C05467=1236.826,137.681,-50.122,-177.956,5.568,148.362
C05468=1236.831,137.432,-50.101,-177.958,5.567,148.362
C05469=1236.835,137.183,-50.081,-177.961,5.566,148.363
C05470=1236.840,136.934,-50.061,-177.963,5.565,148.363
C05471=1236.845,136.684,-50.040,-177.966,5.564,148.364
C05472=1236.849,136.435,-50.019,-177.968,5.562,148.364
C05473=1236.855,136.186,-49.998,-177.971,5.562,148.365
C05474=1236.859,135.937,-49.978,-177.973,5.561,148.365
C05475=1236.864,135.688,-49.957,-177.976,5.560,148.366
C05476=1236.869,135.439,-49.937,-177.979,5.559,148.366
C05477=1236.873,135.190,-49.916,-177.981,5.558,148.367
C05478=1236.878,134.941,-49.895,-177.984,5.557,148.367
C05479=1236.883,134.692,-49.875,-177.986,5.555,148.368
C05480=1236.887,134.443,-49.854,-177.989,5.554,148.368
C05481=1236.893,134.174,-49.833,-177.991,5.554,148.369
C05482=1236.898,133.905,-49.810,-177.994,5.552,148.369
C05483=1236.903,133.636,-49.788,-177.997,5.551,148.370
C05484=1236.908,133.368,-49.767,-178.000,5.550,148.371
C05485=1236.913,133.119,-49.746,-178.002,5.549,148.371
C05486=1236.917,132.870,-49.725,-178.005,5.548,148.372
C05487=1236.922,132.621,-49.705,-178.007,5.548,148.372
C05488=1236.927,132.371,-49.685,-178.010,5.546,148.373
C05489=1236.932,132.122,-49.664,-178.012,5.545,148.373
C05490=1236.936,131.873,-49.644,-178.015,5.544,148.374
C05491=1236.941,131.624,-49.623,-178.018,5.543,148.374
C05492=1236.946,131.375,-49.602,-178.020,5.542,148.375
C05493=1236.951,131.125,-49.583,-178.022,5.541,148.375
C05494=1236.955,130.876,-49.562,-178.025,5.540,148.376
C05495=1236.960,130.627,-49.541,-178.028,5.539,148.376
C05496=1236.965,130.378,-49.521,-178.030,5.538,148.377
C05497=1236.970,130.129,-49.502,-178.032,5.537,148.377
C05498=1236.974,129.880,-49.481,-178.035,5.536,148.378
C05499=1236.979,129.631,-49.461,-178.038,5.535,148.379
C05500=1236.984,129.381,-49.441,-178.040,5.534,148.379
C05501=1236.989,129.132,-49.420,-178.043,5.533,148.380
C05502=1236.993,128.884,-49.400,-178.045,5.532,148.380
C05503=1236.998,128.635,-49.380,-178.048,5.531,148.381
C05504=1237.002,128.385,-49.360,-178.050,5.530,148.381
C05505=1237.008,128.136,-49.339,-178.053,5.529,148.382
C05506=1237.012,127.887,-49.319,-178.056,5.528,148.382
C05507=1237.017,127.638,-49.299,-178.058,5.527,148.383
C05508=1237.022,127.389,-49.279,-178.061,5.526,148.383
C05509=1237.027,127.139,-49.259,-178.063,5.525,148.384
C05510=1237.032,126.890,-49.238,-178.066,5.524,148.384
C05511=1237.036,126.641,-49.218,-178.069,5.523,148.385
C05512=1237.041,126.392,-49.198,-178.071,5.522,148.385
C05513=1237.045,126.143,-49.178,-178.073,5.521,148.386
C05514=1237.051,125.894,-49.159,-178.076,5.520,148.386
C05515=1237.055,125.645,-49.138,-178.078,5.520,148.387
C05516=1237.060,125.396,-49.118,-178.081,5.518,148.388
C05517=1237.064,125.146,-49.098,-178.083,5.517,148.388
C05518=1237.069,124.897,-49.077,-178.086,5.517,148.389
C05519=1237.074,124.648,-49.058,-178.089,5.516,148.389
C05520=1237.079,124.399,-49.038,-178.091,5.514,148.390
C05521=1237.084,124.150,-49.018,-178.094,5.513,148.390
C05522=1237.088,123.901,-48.998,-178.096,5.512,148.391
C05523=1237.093,123.651,-48.978,-178.099,5.512,148.391
C05524=1237.098,123.402,-48.958,-178.101,5.511,148.392
C05525=1237.102,123.153,-48.938,-178.104,5.509,148.392
C05526=1237.107,122.904,-48.918,-178.107,5.509,148.393
C05527=1237.112,122.655,-48.898,-178.109,5.508,148.394
C05528=1237.117,122.406,-48.878,-178.111,5.507,148.394
C05529=1237.121,122.156,-48.858,-178.114,5.506,148.395
C05530=1237.127,121.907,-48.839,-178.117,5.505,148.395
C05531=1237.131,121.659,-48.819,-178.119,5.504,148.396
C05532=1237.136,121.409,-48.799,-178.122,5.503,148.396
C05533=1237.140,121.160,-48.779,-178.124,5.502,148.397
C05534=1237.146,120.910,-48.758,-178.127,5.501,148.397
C05535=1237.151,120.661,-48.739,-178.130,5.500,148.398
C05536=1237.156,120.412,-48.719,-178.132,5.499,148.399
C05537=1237.160,120.163,-48.699,-178.134,5.499,148.399
C05538=1237.164,119.914,-48.679,-178.136,5.498,148.400
C05539=1237.169,119.665,-48.660,-178.140,5.496,148.400
C05540=1237.174,119.416,-48.640,-178.142,5.496,148.401
C05541=1237.179,119.167,-48.620,-178.144,5.495,148.401
C05542=1237.183,118.917,-48.600,-178.147,5.494,148.402
C05543=1237.189,118.668,-48.581,-178.150,5.493,148.403
C05544=1237.193,118.419,-48.561,-178.152,5.492,148.403
C05545=1237.198,118.170,-48.541,-178.155,5.491,148.404
C05546=1237.203,117.920,-48.521,-178.157,5.490,148.404
C05547=1237.208,117.671,-48.502,-178.160,5.489,148.405
C05548=1237.212,117.422,-48.482,-178.162,5.489,148.405
C05549=1237.217,117.173,-48.462,-178.165,5.488,148.406
C05550=1237.222,116.924,-48.443,-178.167,5.486,148.406
C05551=1237.227,116.674,-48.423,-178.170,5.486,148.407
C05552=1237.232,116.425,-48.403,-178.172,5.485,148.407
C05553=1237.237,116.177,-48.383,-178.175,5.484,148.408
C05554=1237.241,115.927,-48.364,-178.177,5.483,148.409
C05555=1237.246,115.678,-48.345,-178.180,5.482,148.409
C05556=1237.250,115.429,-48.324,-178.183,5.481,148.410
C05557=1237.255,115.180,-48.305,-178.185,5.480,148.410
C05558=1237.260,114.930,-48.285,-178.187,5.479,148.411
C05559=1237.265,114.681,-48.266,-178.190,5.479,148.411
C05560=1237.270,114.432,-48.246,-178.193,5.478,148.412
C05561=1237.275,114.182,-48.227,-178.195,5.476,148.412
C05562=1237.279,113.934,-48.207,-178.198,5.476,148.413
C05563=1237.284,113.685,-48.188,-178.201,5.475,148.414
C05564=1237.289,113.435,-48.168,-178.203,5.474,148.414
C05565=1237.294,113.186,-48.149,-178.205,5.473,148.415
C05566=1237.299,112.937,-48.129,-178.208,5.473,148.415
C05567=1237.303,112.688,-48.110,-178.210,5.472,148.416
C05568=1237.308,112.439,-48.091,-178.213,5.470,148.416
C05569=1237.313,112.189,-48.071,-178.216,5.470,148.417
C05570=1237.318,111.940,-48.051,-178.218,5.469,148.417
C05571=1237.323,111.691,-48.032,-178.221,5.468,148.418
C05572=1237.327,111.441,-48.013,-178.223,5.467,148.419
C05573=1237.332,111.193,-47.993,-178.226,5.467,148.419
C05574=1237.337,110.944,-47.973,-178.228,5.465,148.420
C05575=1237.342,110.694,-47.954,-178.231,5.464,148.420
C05576=1237.346,110.446,-47.935,-178.234,5.464,148.421
C05577=1237.351,110.196,-47.915,-178.236,5.463,148.421
C05578=1237.356,109.946,-47.896,-178.238,5.462,148.422
C05579=1237.361,109.698,-47.876,-178.241,5.461,148.423
C05580=1237.365,109.448,-47.857,-178.243,5.460,148.423
C05581=1237.370,109.199,-47.838,-178.246,5.459,148.424
C05582=1237.375,108.950,-47.818,-178.249,5.458,148.424
C05583=1237.381,108.700,-47.800,-178.251,5.457,148.425
C05584=1237.385,108.451,-47.781,-178.254,5.457,148.426
C05585=1237.390,108.182,-47.760,-178.256,5.456,148.426
C05586=1237.395,107.915,-47.739,-178.259,5.455,148.427
C05587=1237.400,107.646,-47.718,-178.262,5.454,148.427
C05588=1237.406,107.378,-47.697,-178.265,5.453,148.428
C05589=1237.411,107.128,-47.678,-178.267,5.452,148.428
C05590=1237.415,106.878,-47.659,-178.269,5.452,148.429
C05591=1237.420,106.630,-47.640,-178.273,5.450,148.430
C05592=1237.425,106.380,-47.620,-178.275,5.450,148.430
C05593=1237.429,106.131,-47.602,-178.277,5.449,148.431
C05594=1237.434,105.882,-47.582,-178.280,5.448,148.431
C05595=1237.439,105.633,-47.563,-178.283,5.447,148.432
C05596=1237.443,105.384,-47.544,-178.285,5.447,148.433
C05597=1237.449,105.134,-47.525,-178.287,5.446,148.433
C05598=1237.453,104.885,-47.506,-178.290,5.445,148.434
C05599=1237.458,104.636,-47.487,-178.293,5.443,148.434
C05600=1237.463,104.387,-47.467,-178.295,5.443,148.435
C05601=1237.468,104.138,-47.448,-178.298,5.442,148.436
C05602=1237.473,103.888,-47.429,-178.300,5.442,148.436
C05603=1237.477,103.639,-47.411,-178.303,5.441,148.437
C05604=1237.482,103.390,-47.391,-178.305,5.440,148.437
C05605=1237.488,103.141,-47.372,-178.308,5.439,148.438
C05606=1237.492,102.891,-47.353,-178.310,5.439,148.439
C05607=1237.497,102.642,-47.334,-178.313,5.438,148.439
C05608=1237.501,102.393,-47.315,-178.316,5.436,148.440
C05609=1237.507,102.144,-47.296,-178.318,5.436,148.440
C05610=1237.511,101.894,-47.277,-178.320,5.435,148.441
C05611=1237.516,101.645,-47.258,-178.323,5.434,148.441
C05612=1237.520,101.396,-47.239,-178.326,5.433,148.442
C05613=1237.526,101.146,-47.220,-178.328,5.433,148.443
C05614=1237.530,100.897,-47.201,-178.330,5.432,148.443
C05615=1237.535,100.648,-47.182,-178.333,5.431,148.444
C05616=1237.540,100.399,-47.164,-178.336,5.431,148.444
C05617=1237.545,100.150,-47.144,-178.338,5.430,148.445
C05618=1237.550,99.901,-47.126,-178.340,5.429,148.445
C05619=1237.555,99.651,-47.107,-178.344,5.428,148.446
C05620=1237.559,99.402,-47.088,-178.346,5.427,148.447
C05621=1237.564,99.153,-47.068,-178.348,5.426,148.447
C05622=1237.569,98.904,-47.050,-178.351,5.425,148.448
C05623=1237.574,98.655,-47.031,-178.354,5.425,148.448
C05624=1237.578,98.405,-47.013,-178.356,5.424,148.449
C05625=1237.584,98.156,-46.994,-178.358,5.423,148.449
C05626=1237.588,97.907,-46.974,-178.361,5.423,148.450
C05627=1237.593,97.657,-46.956,-178.364,5.422,148.451
C05628=1237.597,97.408,-46.937,-178.366,5.421,148.451
C05629=1237.602,97.159,-46.919,-178.368,5.420,148.452
C05630=1237.608,96.910,-46.900,-178.371,5.420,148.452
C05631=1237.612,96.660,-46.881,-178.374,5.418,148.453
C05632=1237.617,96.411,-46.862,-178.377,5.418,148.454
C05633=1237.622,96.162,-46.844,-178.379,5.417,148.454
C05634=1237.627,95.912,-46.824,-178.381,5.416,148.455
C05635=1237.632,95.663,-46.806,-178.384,5.415,148.455
C05636=1237.636,95.414,-46.787,-178.387,5.415,148.456
C05637=1237.642,95.165,-46.769,-178.389,5.414,148.457
C05638=1237.646,94.916,-46.750,-178.391,5.413,148.457
C05639=1237.651,94.666,-46.732,-178.394,5.413,148.458
C05640=1237.656,94.417,-46.712,-178.397,5.412,148.458
C05641=1237.661,94.168,-46.694,-178.399,5.411,148.459
C05642=1237.665,93.919,-46.675,-178.401,5.410,148.460
C05643=1237.670,93.669,-46.657,-178.404,5.410,148.460
C05644=1237.675,93.421,-46.638,-178.407,5.409,148.461
C05645=1237.679,93.171,-46.620,-178.409,5.409,148.461
C05646=1237.685,92.921,-46.601,-178.412,5.407,148.462
C05647=1237.690,92.673,-46.582,-178.415,5.406,148.463
C05648=1237.694,92.423,-46.564,-178.417,5.406,148.463
C05649=1237.700,92.173,-46.545,-178.420,5.405,148.464
C05650=1237.704,91.925,-46.527,-178.422,5.404,148.464
C05651=1237.708,91.675,-46.508,-178.425,5.403,148.465
C05652=1237.714,91.426,-46.489,-178.427,5.403,148.466
C05653=1237.719,91.177,-46.471,-178.430,5.402,148.466
C05654=1237.723,90.927,-46.453,-178.432,5.402,148.467
C05655=1237.728,90.679,-46.434,-178.435,5.401,148.467
C05656=1237.733,90.429,-46.416,-178.437,5.400,148.468
C05657=1237.738,90.179,-46.397,-178.440,5.399,148.469
C05658=1237.743,89.930,-46.379,-178.442,5.399,148.469
C05659=1237.747,89.681,-46.361,-178.445,5.398,148.470
C05660=1237.753,89.432,-46.342,-178.447,5.397,148.470
C05661=1237.757,89.182,-46.324,-178.450,5.397,148.471
C05662=1237.762,88.934,-46.305,-178.452,5.396,148.472
C05663=1237.767,88.684,-46.287,-178.455,5.395,148.472
C05664=1237.772,88.435,-46.268,-178.457,5.394,148.473
C05665=1237.777,88.185,-46.250,-178.460,5.394,148.473
C05666=1237.781,87.936,-46.231,-178.462,5.393,148.474
C05667=1237.786,87.687,-46.213,-178.465,5.393,148.475
C05668=1237.791,87.438,-46.195,-178.468,5.392,148.475
C05669=1237.796,87.188,-46.176,-178.470,5.391,148.476
C05670=1237.801,86.939,-46.158,-178.473,5.389,148.476
C05671=1237.806,86.690,-46.140,-178.476,5.389,148.477
C05672=1237.810,86.441,-46.122,-178.478,5.388,148.478
C05673=1237.815,86.191,-46.103,-178.481,5.388,148.478
C05674=1237.820,85.942,-46.085,-178.483,5.387,148.479
C05675=1237.825,85.692,-46.067,-178.486,5.386,148.479
C05676=1237.830,85.443,-46.049,-178.488,5.385,148.480
C05677=1237.835,85.193,-46.031,-178.491,5.385,148.481
C05678=1237.839,84.945,-46.012,-178.493,5.384,148.481
C05679=1237.844,84.696,-45.994,-178.496,5.383,148.482
C05680=1237.849,84.447,-45.976,-178.498,5.383,148.482
C05681=1237.854,84.197,-45.958,-178.501,5.382,148.483
C05682=1237.858,83.947,-45.940,-178.503,5.381,148.484
C05683=1237.864,83.698,-45.921,-178.506,5.381,148.484
C05684=1237.869,83.449,-45.903,-178.508,5.380,148.485
C05685=1237.874,83.200,-45.885,-178.511,5.379,148.486
C05686=1237.879,82.950,-45.867,-178.513,5.379,148.486
C05687=1237.883,82.701,-45.849,-178.516,5.378,148.487
C05688=1237.888,82.451,-45.831,-178.519,5.377,148.488
C05689=1237.893,82.183,-45.811,-178.521,5.377,148.488
C05690=1237.898,81.915,-45.792,-178.524,5.376,148.489
C05691=1237.904,81.646,-45.772,-178.527,5.376,148.489
C05692=1237.909,81.378,-45.753,-178.529,5.375,148.490
C05693=1237.914,81.129,-45.735,-178.532,5.374,148.491
C05694=1237.919,80.880,-45.717,-178.534,5.373,148.491
C05695=1237.924,80.631,-45.699,-178.537,5.373,148.492
C05696=1237.929,80.381,-45.681,-178.539,5.372,148.493
C05697=1237.933,80.131,-45.662,-178.542,5.372,148.493
C05698=1237.938,79.882,-45.644,-178.544,5.371,148.494
C05699=1237.943,79.633,-45.626,-178.547,5.370,148.495
C05700=1237.948,79.384,-45.608,-178.549,5.369,148.495
C05701=1237.953,79.135,-45.590,-178.552,5.369,148.496
C05702=1237.957,78.886,-45.572,-178.554,5.368,148.496
C05703=1237.962,78.636,-45.554,-178.557,5.368,148.497
C05704=1237.968,78.387,-45.537,-178.560,5.367,148.498
C05705=1237.972,78.137,-45.519,-178.562,5.366,148.498
C05706=1237.977,77.888,-45.501,-178.564,5.366,148.499
C05707=1237.982,77.638,-45.483,-178.567,5.365,148.499
C05708=1237.987,77.389,-45.465,-178.570,5.364,148.500
C05709=1237.992,77.140,-45.447,-178.572,5.364,148.501
C05710=1237.996,76.891,-45.429,-178.575,5.363,148.501
C05711=1238.001,76.642,-45.411,-178.578,5.362,148.502
C05712=1238.007,76.392,-45.394,-178.580,5.362,148.502
C05713=1238.011,76.143,-45.376,-178.582,5.361,148.503
C05714=1238.016,75.894,-45.358,-178.585,5.360,148.504
C05715=1238.021,75.645,-45.340,-178.588,5.360,148.504
C05716=1238.025,75.396,-45.322,-178.590,5.359,148.505
C05717=1238.031,75.146,-45.305,-178.593,5.359,148.506
C05718=1238.035,74.896,-45.287,-178.595,5.358,148.506
C05719=1238.040,74.647,-45.269,-178.598,5.357,148.507
C05720=1238.045,74.397,-45.251,-178.600,5.356,148.507
C05721=1238.050,74.148,-45.233,-178.603,5.356,148.508
C05722=1238.054,73.899,-45.216,-178.606,5.355,148.509
C05723=1238.059,73.650,-45.198,-178.608,5.355,148.509
C05724=1238.064,73.400,-45.180,-178.611,5.354,148.510
C05725=1238.069,73.151,-45.163,-178.613,5.353,148.510
C05726=1238.074,72.902,-45.145,-178.616,5.352,148.511
C05727=1238.079,72.652,-45.127,-178.618,5.352,148.512
C05728=1238.084,72.403,-45.109,-178.621,5.351,148.512
C05729=1238.088,72.154,-45.092,-178.623,5.351,148.513
C05730=1238.093,71.904,-45.074,-178.626,5.350,148.514
C05731=1238.098,71.655,-45.056,-178.628,5.350,148.514
C05732=1238.104,71.406,-45.039,-178.630,5.349,148.515
C05733=1238.108,71.156,-45.021,-178.633,5.349,148.516
C05734=1238.113,70.907,-45.003,-178.636,5.348,148.516
C05735=1238.118,70.658,-44.986,-178.638,5.347,148.517
C05736=1238.123,70.409,-44.968,-178.641,5.347,148.518
C05737=1238.128,70.159,-44.951,-178.643,5.346,148.518
C05738=1238.133,69.910,-44.933,-178.646,5.346,148.519
C05739=1238.137,69.661,-44.916,-178.648,5.345,148.519
C05740=1238.142,69.411,-44.899,-178.651,5.344,148.520
C05741=1238.147,69.162,-44.881,-178.653,5.344,148.521
C05742=1238.152,68.912,-44.863,-178.656,5.343,148.521
C05743=1238.157,68.663,-44.846,-178.659,5.342,148.522
C05744=1238.161,68.414,-44.828,-178.661,5.342,148.523
C05745=1238.167,68.164,-44.811,-178.664,5.341,148.523
C05746=1238.172,67.915,-44.793,-178.667,5.341,148.524
C05747=1238.176,67.665,-44.776,-178.669,5.340,148.524
C05748=1238.181,67.416,-44.758,-178.671,5.339,148.525
C05749=1238.186,67.166,-44.741,-178.673,5.339,148.526
C05750=1238.191,66.918,-44.724,-178.676,5.339,148.526
C05751=1238.196,66.668,-44.706,-178.679,5.338,148.527
C05752=1238.201,66.419,-44.688,-178.681,5.337,148.528
C05753=1238.206,66.170,-44.671,-178.684,5.337,148.528
C05754=1238.211,65.921,-44.654,-178.687,5.336,148.529
C05755=1238.216,65.671,-44.637,-178.689,5.335,148.529
C05756=1238.221,65.422,-44.619,-178.691,5.335,148.530
C05757=1238.225,65.172,-44.602,-178.694,5.334,148.531
C05758=1238.230,64.923,-44.584,-178.697,5.334,148.531
C05759=1238.235,64.673,-44.567,-178.699,5.333,148.532
C05760=1238.240,64.424,-44.550,-178.702,5.332,148.533
C05761=1238.245,64.175,-44.532,-178.704,5.332,148.533
C05762=1238.250,63.925,-44.515,-178.707,5.332,148.534
C05763=1238.255,63.677,-44.498,-178.709,5.331,148.535
C05764=1238.260,63.427,-44.480,-178.711,5.330,148.535
C05765=1238.264,63.177,-44.464,-178.714,5.330,148.536
C05766=1238.269,62.928,-44.446,-178.717,5.329,148.537
C05767=1238.274,62.678,-44.429,-178.719,5.329,148.537
C05768=1238.279,62.429,-44.411,-178.722,5.328,148.538
C05769=1238.284,62.180,-44.394,-178.724,5.328,148.539
C05770=1238.289,61.931,-44.378,-178.727,5.327,148.539
C05771=1238.294,61.682,-44.360,-178.730,5.326,148.540
C05772=1238.299,61.432,-44.342,-178.732,5.326,148.541
C05773=1238.304,61.182,-44.326,-178.735,5.325,148.541
C05774=1238.308,60.933,-44.308,-178.737,5.325,148.542
C05775=1238.313,60.684,-44.291,-178.739,5.324,148.542
C05776=1238.318,60.434,-44.274,-178.742,5.324,148.543
C05777=1238.323,60.185,-44.257,-178.744,5.323,148.544
C05778=1238.328,59.936,-44.239,-178.747,5.323,148.544
C05779=1238.333,59.686,-44.222,-178.750,5.322,148.545
C05780=1238.338,59.437,-44.206,-178.752,5.321,148.546
C05781=1238.343,59.188,-44.188,-178.755,5.321,148.546
C05782=1238.347,58.938,-44.171,-178.758,5.320,148.547
C05783=1238.353,58.689,-44.154,-178.760,5.320,148.548
C05784=1238.358,58.440,-44.137,-178.762,5.320,148.548
C05785=1238.363,58.190,-44.120,-178.764,5.319,148.549
C05786=1238.367,57.941,-44.103,-178.767,5.318,148.549
C05787=1238.372,57.691,-44.085,-178.770,5.318,148.550
C05788=1238.377,57.442,-44.069,-178.772,5.317,148.551
C05789=1238.382,57.192,-44.052,-178.775,5.317,148.551
C05790=1238.387,56.943,-44.035,-178.778,5.316,148.552
C05791=1238.392,56.694,-44.017,-178.780,5.315,148.553
C05792=1238.396,56.444,-44.001,-178.783,5.315,148.553
C05793=1238.402,56.176,-43.982,-178.786,5.314,148.554
C05794=1238.407,55.908,-43.964,-178.788,5.314,148.555
C05795=1238.413,55.639,-43.946,-178.791,5.313,148.555
C05796=1238.418,55.371,-43.928,-178.793,5.313,148.556
C05797=1238.423,55.121,-43.910,-178.796,5.312,148.557
C05798=1238.428,54.872,-43.894,-178.798,5.312,148.557
C05799=1238.432,54.623,-43.877,-178.801,5.312,148.558
C05800=1238.438,54.373,-43.860,-178.803,5.311,148.559
C05801=1238.442,54.124,-43.844,-178.806,5.310,148.559
C05802=1238.448,53.874,-43.827,-178.809,5.310,148.560
C05803=1238.452,53.625,-43.810,-178.811,5.309,148.561
C05804=1238.457,53.376,-43.793,-178.814,5.309,148.561
C05805=1238.462,53.126,-43.775,-178.817,5.308,148.562
C05806=1238.467,52.878,-43.759,-178.819,5.308,148.563
C05807=1238.472,52.628,-43.742,-178.821,5.307,148.563
C05808=1238.477,52.378,-43.725,-178.823,5.307,148.564
C05809=1238.482,52.129,-43.709,-178.826,5.306,148.565
C05810=1238.487,51.880,-43.691,-178.829,5.306,148.565
C05811=1238.491,51.630,-43.675,-178.831,5.305,148.566
C05812=1238.496,51.381,-43.658,-178.834,5.305,148.567
C05813=1238.502,51.132,-43.641,-178.836,5.305,148.567
C05814=1238.506,50.882,-43.625,-178.839,5.304,148.568
C05815=1238.511,50.633,-43.608,-178.841,5.304,148.569
C05816=1238.516,50.384,-43.591,-178.844,5.303,148.569
C05817=1238.521,50.134,-43.574,-178.847,5.302,148.570
C05818=1238.525,49.885,-43.558,-178.849,5.302,148.571
C05819=1238.531,49.635,-43.541,-178.852,5.301,148.571
C05820=1238.536,49.385,-43.525,-178.854,5.302,148.572
C05821=1238.540,49.136,-43.508,-178.857,5.301,148.573
C05822=1238.546,48.887,-43.491,-178.859,5.300,148.573
C05823=1238.551,48.637,-43.475,-178.861,5.299,148.574
C05824=1238.555,48.388,-43.458,-178.864,5.299,148.574
C05825=1238.560,48.139,-43.442,-178.867,5.298,148.575
C05826=1238.566,47.889,-43.424,-178.869,5.298,148.576
C05827=1238.570,47.640,-43.408,-178.871,5.298,148.576
C05828=1238.575,47.391,-43.391,-178.874,5.297,148.577
C05829=1238.580,47.141,-43.375,-178.877,5.297,148.578
C05830=1238.585,46.891,-43.358,-178.879,5.296,148.578
C05831=1238.590,46.642,-43.342,-178.882,5.296,148.579
C05832=1238.595,46.393,-43.325,-178.885,5.295,148.580
C05833=1238.599,46.143,-43.309,-178.887,5.295,148.580
C05834=1238.605,45.894,-43.292,-178.889,5.295,148.581
C05835=1238.610,45.644,-43.276,-178.892,5.294,148.582
C05836=1238.615,45.395,-43.259,-178.895,5.294,148.582
C05837=1238.619,45.146,-43.243,-178.897,5.293,148.583
C05838=1238.624,44.896,-43.226,-178.900,5.292,148.584
C05839=1238.630,44.647,-43.209,-178.902,5.292,148.584
C05840=1238.634,44.397,-43.193,-178.905,5.292,148.585
C05841=1238.639,44.148,-43.177,-178.907,5.291,148.586
C05842=1238.644,43.899,-43.160,-178.910,5.291,148.586
C05843=1238.648,43.649,-43.144,-178.912,5.290,148.587
C05844=1238.655,43.400,-43.127,-178.915,5.289,148.588
C05845=1238.659,43.150,-43.111,-178.917,5.289,148.588
C05846=1238.664,42.901,-43.094,-178.919,5.289,148.589
C05847=1238.669,42.652,-43.078,-178.922,5.288,148.590
C05848=1238.673,42.402,-43.062,-178.925,5.288,148.590
C05849=1238.678,42.153,-43.045,-178.927,5.287,148.591
C05850=1238.683,41.904,-43.029,-178.930,5.287,148.592
C05851=1238.689,41.654,-43.013,-178.932,5.287,148.592
C05852=1238.694,41.404,-42.996,-178.935,5.286,148.593
C05853=1238.699,41.156,-42.980,-178.937,5.286,148.594
C05854=1238.703,40.906,-42.964,-178.940,5.285,148.594
C05855=1238.708,40.656,-42.947,-178.942,5.285,148.595
C05856=1238.713,40.407,-42.931,-178.945,5.284,148.596
C05857=1238.718,40.157,-42.915,-178.947,5.284,148.596
C05858=1238.723,39.908,-42.898,-178.950,5.284,148.597
C05859=1238.727,39.659,-42.882,-178.952,5.283,148.598
C05860=1238.733,39.409,-42.866,-178.955,5.283,148.598
C05861=1238.738,39.160,-42.849,-178.958,5.282,148.599
C05862=1238.743,38.910,-42.833,-178.960,5.282,148.600
C05863=1238.748,38.661,-42.817,-178.962,5.282,148.600
C05864=1238.753,38.411,-42.801,-178.965,5.281,148.601
C05865=1238.758,38.162,-42.784,-178.968,5.281,148.602
C05866=1238.763,37.913,-42.768,-178.970,5.280,148.602
C05867=1238.768,37.663,-42.752,-178.973,5.279,148.603
C05868=1238.773,37.414,-42.736,-178.975,5.280,148.604
C05869=1238.777,37.164,-42.720,-178.978,5.279,148.604
C05870=1238.782,36.915,-42.704,-178.980,5.279,148.605
C05871=1238.787,36.665,-42.688,-178.983,5.278,148.606
C05872=1238.792,36.416,-42.671,-178.986,5.277,148.606
C05873=1238.797,36.166,-42.655,-178.988,5.278,148.607
C05874=1238.802,35.918,-42.639,-178.990,5.277,148.608
C05875=1238.807,35.667,-42.623,-178.993,5.277,148.609
C05876=1238.812,35.419,-42.607,-178.996,5.276,148.609
C05877=1238.817,35.169,-42.591,-178.998,5.275,148.610
C05878=1238.822,34.920,-42.575,-179.000,5.276,148.611
C05879=1238.827,34.670,-42.559,-179.003,5.275,148.611
C05880=1238.832,34.421,-42.542,-179.006,5.275,148.612
C05881=1238.837,34.171,-42.526,-179.008,5.274,148.613
C05882=1238.842,33.921,-42.511,-179.011,5.273,148.613
C05883=1238.847,33.673,-42.494,-179.013,5.273,148.614
C05884=1238.852,33.423,-42.479,-179.015,5.273,148.614
C05885=1238.857,33.174,-42.462,-179.018,5.272,148.615
C05886=1238.862,32.924,-42.446,-179.020,5.272,148.616
C05887=1238.866,32.675,-42.431,-179.023,5.272,148.616
C05888=1238.871,32.425,-42.415,-179.025,5.271,148.617
C05889=1238.876,32.176,-42.399,-179.028,5.271,148.618
C05890=1238.881,31.927,-42.383,-179.030,5.270,148.618
C05891=1238.886,31.677,-42.367,-179.033,5.270,148.619
C05892=1238.891,31.427,-42.351,-179.035,5.270,148.620
C05893=1238.896,31.178,-42.334,-179.038,5.269,148.621
C05894=1238.901,30.928,-42.319,-179.040,5.269,148.621
C05895=1238.907,30.679,-42.303,-179.043,5.268,148.622
C05896=1238.911,30.430,-42.287,-179.046,5.268,148.623
C05897=1238.916,30.161,-42.270,-179.048,5.268,148.623
C05898=1238.922,29.893,-42.253,-179.051,5.268,148.624
C05899=1238.927,29.624,-42.236,-179.054,5.267,148.625
C05900=1238.932,29.355,-42.219,-179.056,5.267,148.625
C05901=1238.937,29.106,-42.203,-179.059,5.266,148.626
C05902=1238.942,28.856,-42.187,-179.062,5.265,148.627
C05903=1238.947,28.607,-42.171,-179.064,5.265,148.628
C05904=1238.953,28.358,-42.155,-179.066,5.265,148.628
C05905=1238.957,28.108,-42.140,-179.069,5.265,148.629
C05906=1238.962,27.858,-42.124,-179.072,5.264,148.630
C05907=1238.967,27.610,-42.108,-179.074,5.263,148.630
C05908=1238.972,27.360,-42.092,-179.076,5.264,148.631
C05909=1238.977,27.110,-42.077,-179.079,5.263,148.632
C05910=1238.982,26.861,-42.062,-179.082,5.263,148.632
C05911=1238.987,26.612,-42.045,-179.084,5.262,148.633
C05912=1238.992,26.362,-42.029,-179.086,5.262,148.634
C05913=1238.997,26.113,-42.014,-179.089,5.262,148.634
C05914=1239.001,25.863,-41.998,-179.092,5.261,148.635
C05915=1239.007,25.614,-41.983,-179.094,5.261,148.636
C05916=1239.012,25.364,-41.967,-179.096,5.261,148.636
C05917=1239.017,25.115,-41.951,-179.099,5.260,148.637
C05918=1239.022,24.865,-41.935,-179.102,5.260,148.638
C05919=1239.027,24.616,-41.920,-179.104,5.259,148.638
C05920=1239.031,24.366,-41.904,-179.106,5.259,148.639
C05921=1239.037,24.117,-41.888,-179.109,5.259,148.640
C05922=1239.041,23.868,-41.873,-179.112,5.259,148.641
C05923=1239.046,23.617,-41.857,-179.115,5.258,148.641
C05924=1239.052,23.368,-41.842,-179.117,5.257,148.642
C05925=1239.057,23.119,-41.826,-179.119,5.258,148.643
C05926=1239.061,22.869,-41.810,-179.122,5.257,148.643
C05927=1239.066,22.620,-41.795,-179.125,5.257,148.644
C05928=1239.072,22.371,-41.779,-179.127,5.256,148.645
C05929=1239.076,22.122,-41.764,-179.129,5.256,148.645
C05930=1239.081,21.871,-41.748,-179.132,5.256,148.646
C05931=1239.086,21.622,-41.733,-179.135,5.255,148.647
C05932=1239.091,21.373,-41.718,-179.137,5.255,148.647
C05933=1239.096,21.124,-41.702,-179.139,5.255,148.648
C05934=1239.101,20.873,-41.686,-179.142,5.254,148.649
C05935=1239.106,20.624,-41.671,-179.145,5.254,148.650
C05936=1239.111,20.375,-41.655,-179.147,5.254,148.650
C05937=1239.116,20.125,-41.639,-179.149,5.254,148.651
C05938=1239.121,19.876,-41.624,-179.152,5.253,148.652
C05939=1239.126,19.626,-41.609,-179.155,5.252,148.652
C05940=1239.131,19.377,-41.593,-179.157,5.253,148.653
C05941=1239.136,19.128,-41.578,-179.159,5.252,148.654
C05942=1239.141,18.878,-41.562,-179.162,5.252,148.654
C05943=1239.146,18.628,-41.547,-179.165,5.251,148.655
C05944=1239.151,18.379,-41.532,-179.167,5.251,148.656
C05945=1239.156,18.130,-41.516,-179.170,5.251,148.656
C05946=1239.160,17.880,-41.501,-179.172,5.250,148.657
C05947=1239.166,17.631,-41.485,-179.175,5.250,148.658
C05948=1239.171,17.381,-41.471,-179.177,5.250,148.658
C05949=1239.176,17.132,-41.455,-179.180,5.249,148.659
C05950=1239.181,16.882,-41.440,-179.182,5.249,148.660
C05951=1239.186,16.632,-41.424,-179.185,5.248,148.660
C05952=1239.191,16.383,-41.409,-179.187,5.248,148.661
C05953=1239.196,16.134,-41.394,-179.190,5.248,148.662
C05954=1239.201,15.885,-41.378,-179.192,5.247,148.663
C05955=1239.206,15.635,-41.363,-179.194,5.248,148.663
C05956=1239.211,15.385,-41.348,-179.197,5.247,148.664
C05957=1239.216,15.135,-41.332,-179.200,5.247,148.665
C05958=1239.221,14.886,-41.317,-179.202,5.246,148.665
C05959=1239.226,14.637,-41.302,-179.204,5.246,148.666
C05960=1239.231,14.388,-41.287,-179.207,5.246,148.667
C05961=1239.236,14.138,-41.271,-179.210,5.246,148.668
C05962=1239.240,13.888,-41.257,-179.212,5.246,148.668
C05963=1239.246,13.638,-41.241,-179.215,5.245,148.669
C05964=1239.251,13.389,-41.226,-179.217,5.245,148.670
C05965=1239.256,13.140,-41.210,-179.220,5.244,148.670
C05966=1239.261,12.890,-41.196,-179.222,5.244,148.671
C05967=1239.266,12.641,-41.181,-179.225,5.244,148.672
C05968=1239.270,12.391,-41.165,-179.227,5.243,148.672
C05969=1239.276,12.142,-41.150,-179.230,5.244,148.673
C05970=1239.281,11.892,-41.135,-179.232,5.243,148.674
C05971=1239.285,11.643,-41.120,-179.235,5.242,148.674
C05972=1239.291,11.393,-41.105,-179.238,5.242,148.675
C05973=1239.295,11.144,-41.090,-179.240,5.242,148.676
C05974=1239.301,10.894,-41.075,-179.242,5.242,148.676
C05975=1239.306,10.645,-41.060,-179.245,5.241,148.677
C05976=1239.310,10.395,-41.044,-179.247,5.241,148.678
C05977=1239.315,10.145,-41.030,-179.250,5.241,148.679
C05978=1239.321,9.896,-41.014,-179.252,5.240,148.679
C05979=1239.325,9.647,-40.999,-179.255,5.240,148.680
C05980=1239.330,9.397,-40.985,-179.257,5.240,148.681
C05981=1239.336,9.148,-40.969,-179.260,5.239,148.681
C05982=1239.340,8.899,-40.954,-179.262,5.239,148.682
C05983=1239.346,8.649,-40.939,-179.265,5.240,148.683
C05984=1239.351,8.400,-40.924,-179.268,5.239,148.684
C05985=1239.355,8.151,-40.909,-179.270,5.238,148.684
C05986=1239.361,7.901,-40.895,-179.272,5.239,148.685
C05987=1239.365,7.651,-40.879,-179.275,5.238,148.686
C05988=1239.370,7.401,-40.865,-179.278,5.238,148.686
C05989=1239.376,7.152,-40.849,-179.280,5.237,148.687
C05990=1239.380,6.903,-40.834,-179.282,5.237,148.688
C05991=1239.385,6.653,-40.820,-179.285,5.237,148.688
C05992=1239.391,6.403,-40.804,-179.288,5.236,148.689
C05993=1239.395,6.154,-40.790,-179.290,5.237,148.690
C05994=1239.400,5.905,-40.775,-179.292,5.236,148.690
C05995=1239.406,5.655,-40.760,-179.295,5.235,148.691
C05996=1239.410,5.406,-40.745,-179.297,5.236,148.692
C05997=1239.415,5.156,-40.730,-179.300,5.235,148.692
C05998=1239.421,4.906,-40.715,-179.302,5.235,148.693
C05999=1239.425,4.657,-40.700,-179.304,5.235,148.694
C06000=1239.430,4.408,-40.686,-179.307,5.234,148.695
C06001=1239.436,4.138,-40.670,-179.310,5.234,148.695
C06002=1239.441,3.870,-40.654,-179.313,5.234,148.696
C06003=1239.447,3.601,-40.638,-179.316,5.233,148.697
C06004=1239.452,3.332,-40.622,-179.318,5.234,148.698
C06005=1239.457,3.083,-40.607,-179.321,5.233,148.698
C06006=1239.462,2.833,-40.593,-179.323,5.233,148.699
C06007=1239.467,2.584,-40.577,-179.325,5.233,148.700
C06008=1239.472,2.334,-40.563,-179.328,5.232,148.701
C06009=1239.477,2.085,-40.548,-179.331,5.232,148.701
C06010=1239.482,1.835,-40.534,-179.333,5.231,148.702
C06011=1239.488,1.585,-40.519,-179.336,5.232,148.703
C06012=1239.492,1.336,-40.504,-179.338,5.231,148.703
C06013=1239.497,1.086,-40.490,-179.341,5.231,148.704
C06014=1239.502,0.837,-40.475,-179.343,5.231,148.705
C06015=1239.508,0.587,-40.460,-179.346,5.230,148.705
C06016=1239.513,0.337,-40.445,-179.348,5.230,148.706
C06017=1239.517,0.088,-40.430,-179.350,5.230,148.707
C06018=1239.522,-0.161,-40.416,-179.353,5.229,148.707
C06019=1239.527,-0.410,-40.401,-179.356,5.229,148.708
C06020=1239.532,-0.660,-40.386,-179.358,5.230,148.709
C06021=1239.537,-0.910,-40.372,-179.361,5.229,148.710
C06022=1239.542,-1.159,-40.357,-179.363,5.228,148.710
C06023=1239.547,-1.409,-40.343,-179.366,5.229,148.711
C06024=1239.552,-1.659,-40.328,-179.368,5.228,148.712
C06025=1239.557,-1.907,-40.314,-179.371,5.228,148.712
C06026=1239.563,-2.157,-40.299,-179.373,5.228,148.713
C06027=1239.568,-2.407,-40.285,-179.376,5.227,148.714
C06028=1239.573,-2.657,-40.270,-179.378,5.227,148.715
C06029=1239.577,-2.906,-40.255,-179.380,5.227,148.715
C06030=1239.582,-3.155,-40.241,-179.383,5.227,148.716
C06031=1239.587,-3.405,-40.227,-179.386,5.226,148.717
C06032=1239.592,-3.654,-40.212,-179.388,5.226,148.717
C06033=1239.598,-3.904,-40.197,-179.390,5.226,148.718
C06034=1239.603,-4.154,-40.183,-179.394,5.226,148.719
C06035=1239.608,-4.404,-40.168,-179.396,5.226,148.720
C06036=1239.613,-4.653,-40.154,-179.398,5.225,148.720
C06037=1239.618,-4.902,-40.140,-179.401,5.225,148.721
C06038=1239.623,-5.151,-40.125,-179.403,5.225,148.722
C06039=1239.628,-5.401,-40.111,-179.406,5.225,148.722
C06040=1239.633,-5.651,-40.097,-179.408,5.225,148.723
C06041=1239.637,-5.900,-40.082,-179.410,5.224,148.724
C06042=1239.642,-6.150,-40.067,-179.413,5.224,148.724
C06043=1239.647,-6.399,-40.053,-179.415,5.224,148.725
C06044=1239.653,-6.649,-40.038,-179.418,5.224,148.726
C06045=1239.658,-6.899,-40.024,-179.420,5.223,148.727
C06046=1239.663,-7.148,-40.010,-179.422,5.223,148.727
C06047=1239.668,-7.397,-39.995,-179.425,5.223,148.728
C06048=1239.673,-7.647,-39.981,-179.428,5.223,148.729
C06049=1239.678,-7.897,-39.967,-179.430,5.223,148.730
C06050=1239.683,-8.146,-39.952,-179.433,5.222,148.730
C06051=1239.688,-8.396,-39.938,-179.436,5.222,148.731
C06052=1239.693,-8.646,-39.924,-179.438,5.222,148.732
C06053=1239.698,-8.895,-39.910,-179.440,5.222,148.732
C06054=1239.703,-9.144,-39.896,-179.443,5.221,148.733
C06055=1239.708,-9.394,-39.881,-179.445,5.221,148.734
C06056=1239.713,-9.643,-39.866,-179.448,5.221,148.734
C06057=1239.718,-9.893,-39.852,-179.450,5.220,148.735
C06058=1239.723,-10.143,-39.838,-179.453,5.221,148.736
C06059=1239.728,-10.392,-39.824,-179.455,5.220,148.736
C06060=1239.733,-10.641,-39.810,-179.457,5.220,148.737
C06061=1239.738,-10.891,-39.795,-179.460,5.220,148.738
C06062=1239.743,-11.141,-39.781,-179.463,5.220,148.739
C06063=1239.748,-11.390,-39.767,-179.465,5.220,148.739
C06064=1239.754,-11.639,-39.753,-179.468,5.219,148.740
C06065=1239.759,-11.889,-39.739,-179.470,5.219,148.741
C06066=1239.764,-12.139,-39.724,-179.473,5.219,148.742
C06067=1239.768,-12.388,-39.711,-179.475,5.219,148.742
C06068=1239.773,-12.638,-39.696,-179.478,5.218,148.743
C06069=1239.778,-12.887,-39.682,-179.480,5.218,148.744
C06070=1239.783,-13.137,-39.668,-179.483,5.218,148.744
C06071=1239.788,-13.386,-39.654,-179.485,5.218,148.745
C06072=1239.793,-13.636,-39.640,-179.487,5.218,148.746
C06073=1239.799,-13.885,-39.626,-179.491,5.218,148.747
C06074=1239.804,-14.135,-39.611,-179.493,5.218,148.747
C06075=1239.809,-14.385,-39.597,-179.495,5.217,148.748
C06076=1239.814,-14.634,-39.583,-179.498,5.217,148.749
C06077=1239.819,-14.884,-39.569,-179.500,5.217,148.749
C06078=1239.824,-15.133,-39.556,-179.503,5.217,148.750
C06079=1239.829,-15.383,-39.542,-179.505,5.217,148.751
C06080=1239.834,-15.633,-39.527,-179.507,5.216,148.751
C06081=1239.839,-15.882,-39.513,-179.510,5.216,148.752
C06082=1239.844,-16.131,-39.499,-179.512,5.216,148.753
C06083=1239.849,-16.381,-39.485,-179.515,5.216,148.754
C06084=1239.854,-16.631,-39.471,-179.517,5.215,148.754
C06085=1239.859,-16.880,-39.457,-179.520,5.216,148.755
C06086=1239.864,-17.130,-39.444,-179.523,5.215,148.756
C06087=1239.869,-17.380,-39.429,-179.525,5.215,148.757
C06088=1239.874,-17.629,-39.415,-179.527,5.215,148.757
C06089=1239.880,-17.878,-39.401,-179.530,5.214,148.758
C06090=1239.885,-18.128,-39.387,-179.532,5.215,148.759
C06091=1239.889,-18.377,-39.373,-179.535,5.214,148.759
C06092=1239.895,-18.627,-39.360,-179.537,5.214,148.760
C06093=1239.900,-18.877,-39.346,-179.540,5.214,148.761
C06094=1239.905,-19.127,-39.332,-179.542,5.213,148.761
C06095=1239.910,-19.376,-39.317,-179.544,5.214,148.762
C06096=1239.914,-19.625,-39.304,-179.547,5.213,148.763
C06097=1239.920,-19.875,-39.290,-179.550,5.213,148.764
C06098=1239.925,-20.125,-39.276,-179.552,5.213,148.764
C06099=1239.930,-20.374,-39.262,-179.555,5.213,148.765
C06100=1239.935,-20.624,-39.248,-179.557,5.213,148.766
C06101=1239.940,-20.874,-39.235,-179.560,5.213,148.767
C06102=1239.945,-21.123,-39.221,-179.562,5.212,148.767
C06103=1239.950,-21.372,-39.207,-179.564,5.212,148.768
C06104=1239.955,-21.622,-39.193,-179.567,5.212,148.769
C06105=1239.960,-21.891,-39.178,-179.570,5.212,148.770
C06106=1239.966,-22.160,-39.164,-179.572,5.212,148.770
C06107=1239.971,-22.429,-39.149,-179.575,5.211,148.771
C06108=1239.977,-22.699,-39.134,-179.578,5.211,148.772
C06109=1239.983,-22.948,-39.120,-179.580,5.212,148.773
C06110=1239.987,-23.198,-39.107,-179.583,5.211,148.773
C06111=1239.992,-23.448,-39.092,-179.585,5.211,148.774
C06112=1239.998,-23.697,-39.079,-179.588,5.211,148.775
C06113=1240.003,-23.947,-39.065,-179.590,5.210,148.775
C06114=1240.007,-24.196,-39.051,-179.592,5.211,148.776
C06115=1240.013,-24.446,-39.038,-179.595,5.210,148.777
C06116=1240.018,-24.696,-39.024,-179.598,5.210,148.777
C06117=1240.022,-24.944,-39.010,-179.600,5.210,148.778
C06118=1240.028,-25.195,-38.997,-179.602,5.209,148.779
C06119=1240.033,-25.444,-38.983,-179.605,5.210,148.780
C06120=1240.038,-25.694,-38.970,-179.608,5.209,148.780
C06121=1240.043,-25.943,-38.956,-179.610,5.209,148.781
C06122=1240.048,-26.192,-38.942,-179.612,5.209,148.782
C06123=1240.053,-26.442,-38.929,-179.615,5.209,148.783
C06124=1240.058,-26.692,-38.915,-179.617,5.209,148.783
C06125=1240.063,-26.941,-38.902,-179.620,5.209,148.784
C06126=1240.068,-27.191,-38.888,-179.622,5.208,148.785
C06127=1240.074,-27.441,-38.874,-179.624,5.208,148.785
C06128=1240.078,-27.690,-38.861,-179.627,5.208,148.786
C06129=1240.083,-27.940,-38.847,-179.629,5.208,148.787
C06130=1240.089,-28.190,-38.833,-179.632,5.208,148.788
C06131=1240.093,-28.439,-38.820,-179.635,5.207,148.788
C06132=1240.099,-28.689,-38.806,-179.637,5.208,148.789
C06133=1240.103,-28.938,-38.793,-179.640,5.207,148.790
C06134=1240.109,-29.188,-38.780,-179.642,5.208,148.790
C06135=1240.113,-29.437,-38.766,-179.645,5.207,148.791
C06136=1240.118,-29.687,-38.752,-179.647,5.207,148.792
C06137=1240.124,-29.936,-38.738,-179.649,5.207,148.793
C06138=1240.128,-30.186,-38.725,-179.652,5.206,148.793
C06139=1240.134,-30.436,-38.712,-179.654,5.207,148.794
C06140=1240.139,-30.685,-38.699,-179.657,5.206,148.795
C06141=1240.144,-30.935,-38.685,-179.659,5.207,148.796
C06142=1240.149,-31.184,-38.672,-179.662,5.206,148.796
C06143=1240.154,-31.434,-38.658,-179.665,5.206,148.797
C06144=1240.159,-31.683,-38.645,-179.667,5.206,148.798
C06145=1240.165,-31.933,-38.632,-179.669,5.206,148.798
C06146=1240.169,-32.183,-38.619,-179.671,5.206,148.799
C06147=1240.175,-32.432,-38.605,-179.674,5.205,148.800
C06148=1240.180,-32.682,-38.591,-179.676,5.206,148.800
C06149=1240.185,-32.931,-38.578,-179.679,5.205,148.801
C06150=1240.190,-33.181,-38.564,-179.681,5.205,148.802
C06151=1240.195,-33.431,-38.552,-179.684,5.205,148.803
C06152=1240.200,-33.680,-38.537,-179.687,5.205,148.803
C06153=1240.205,-33.930,-38.525,-179.689,5.205,148.804
C06154=1240.210,-34.180,-38.512,-179.691,5.205,148.805
C06155=1240.215,-34.429,-38.498,-179.694,5.205,148.806
C06156=1240.220,-34.679,-38.485,-179.696,5.204,148.806
C06157=1240.226,-34.928,-38.472,-179.699,5.204,148.807
C06158=1240.230,-35.178,-38.458,-179.701,5.204,148.808
C06159=1240.236,-35.427,-38.445,-179.704,5.204,148.808
C06160=1240.240,-35.677,-38.432,-179.706,5.204,148.809
C06161=1240.246,-35.926,-38.418,-179.708,5.203,148.810
C06162=1240.250,-36.177,-38.405,-179.712,5.203,148.811
C06163=1240.256,-36.426,-38.392,-179.714,5.204,148.811
C06164=1240.260,-36.676,-38.378,-179.716,5.203,148.812
C06165=1240.266,-36.925,-38.366,-179.718,5.203,148.813
C06166=1240.271,-37.174,-38.352,-179.721,5.203,148.814
C06167=1240.276,-37.425,-38.339,-179.723,5.203,148.814
C06168=1240.281,-37.674,-38.326,-179.726,5.203,148.815
C06169=1240.286,-37.924,-38.313,-179.728,5.203,148.816
C06170=1240.292,-38.173,-38.299,-179.731,5.202,148.816
C06171=1240.296,-38.423,-38.286,-179.733,5.202,148.817
C06172=1240.301,-38.672,-38.273,-179.736,5.203,148.818
C06173=1240.307,-38.922,-38.260,-179.738,5.202,148.819
C06174=1240.312,-39.172,-38.247,-179.741,5.202,148.819
C06175=1240.317,-39.421,-38.234,-179.743,5.202,148.820
C06176=1240.322,-39.671,-38.221,-179.745,5.202,148.821
C06177=1240.327,-39.920,-38.208,-179.748,5.202,148.821
C06178=1240.332,-40.170,-38.194,-179.751,5.201,148.822
C06179=1240.337,-40.420,-38.181,-179.753,5.202,148.823
C06180=1240.342,-40.669,-38.169,-179.755,5.201,148.824
C06181=1240.348,-40.919,-38.155,-179.757,5.201,148.824
C06182=1240.353,-41.168,-38.142,-179.761,5.201,148.825
C06183=1240.357,-41.419,-38.130,-179.763,5.202,148.826
C06184=1240.363,-41.668,-38.116,-179.765,5.201,148.827
C06185=1240.368,-41.917,-38.103,-179.767,5.201,148.827
C06186=1240.372,-42.167,-38.090,-179.770,5.201,148.828
C06187=1240.378,-42.416,-38.077,-179.773,5.200,148.829
C06188=1240.383,-42.666,-38.064,-179.775,5.201,148.829
C06189=1240.388,-42.916,-38.051,-179.778,5.200,148.830
C06190=1240.393,-43.165,-38.039,-179.780,5.200,148.831
C06191=1240.398,-43.415,-38.025,-179.782,5.200,148.831
C06192=1240.403,-43.665,-38.013,-179.784,5.200,148.832
C06193=1240.409,-43.914,-38.000,-179.788,5.200,148.833
C06194=1240.413,-44.163,-37.986,-179.790,5.200,148.834
C06195=1240.419,-44.413,-37.973,-179.792,5.200,148.835
C06196=1240.424,-44.662,-37.960,-179.795,5.199,148.835
C06197=1240.428,-44.912,-37.947,-179.797,5.200,148.836
C06198=1240.434,-45.162,-37.934,-179.800,5.199,148.837
C06199=1240.439,-45.411,-37.922,-179.802,5.200,148.837
C06200=1240.444,-45.661,-37.909,-179.804,5.199,148.838
C06201=1240.449,-45.911,-37.896,-179.807,5.199,148.839
C06202=1240.454,-46.160,-37.884,-179.809,5.199,148.839
C06203=1240.459,-46.410,-37.870,-179.812,5.200,148.840
C06204=1240.464,-46.660,-37.857,-179.814,5.199,148.841
C06205=1240.470,-46.909,-37.845,-179.817,5.199,148.842
C06206=1240.474,-47.159,-37.832,-179.819,5.199,148.842
C06207=1240.480,-47.409,-37.819,-179.822,5.198,148.843
C06208=1240.485,-47.658,-37.806,-179.824,5.199,148.844
C06209=1240.490,-47.928,-37.792,-179.827,5.198,148.845
C06210=1240.496,-48.198,-37.778,-179.829,5.199,148.846
C06211=1240.501,-48.467,-37.765,-179.832,5.198,148.846
C06212=1240.506,-48.737,-37.751,-179.835,5.198,148.847
C06213=1240.513,-48.987,-37.739,-179.837,5.198,148.848
C06214=1240.518,-49.236,-37.726,-179.840,5.198,148.849
C06215=1240.522,-49.486,-37.713,-179.842,5.198,148.849
C06216=1240.527,-49.735,-37.700,-179.845,5.198,148.850
C06217=1240.532,-49.985,-37.688,-179.847,5.198,148.851
C06218=1240.537,-50.235,-37.675,-179.849,5.198,148.851
C06219=1240.543,-50.484,-37.662,-179.852,5.197,148.852
C06220=1240.548,-50.734,-37.649,-179.854,5.198,148.853
C06221=1240.553,-50.983,-37.636,-179.857,5.197,148.853
C06222=1240.558,-51.234,-37.624,-179.859,5.197,148.854
C06223=1240.563,-51.483,-37.612,-179.861,5.197,148.855
C06224=1240.568,-51.732,-37.599,-179.864,5.198,148.856
C06225=1240.573,-51.982,-37.586,-179.867,5.197,148.857
C06226=1240.578,-52.232,-37.573,-179.869,5.197,148.857
C06227=1240.584,-52.481,-37.560,-179.871,5.197,148.858
C06228=1240.589,-52.731,-37.548,-179.874,5.197,148.859
C06229=1240.594,-52.981,-37.536,-179.876,5.197,148.859
C06230=1240.599,-53.231,-37.523,-179.878,5.197,148.860
C06231=1240.604,-53.480,-37.510,-179.881,5.197,148.861
C06232=1240.609,-53.729,-37.498,-179.883,5.197,148.861
C06233=1240.614,-53.979,-37.486,-179.886,5.196,148.862
C06234=1240.620,-54.228,-37.473,-179.888,5.196,148.863
C06235=1240.624,-54.478,-37.460,-179.891,5.197,148.864
C06236=1240.629,-54.728,-37.447,-179.894,5.196,148.865
C06237=1240.635,-54.978,-37.436,-179.896,5.196,148.865
C06238=1240.640,-55.227,-37.423,-179.898,5.196,148.866
C06239=1240.644,-55.477,-37.410,-179.900,5.196,148.867
C06240=1240.649,-55.726,-37.397,-179.903,5.196,148.867
C06241=1240.655,-55.976,-37.386,-179.905,5.196,148.868
C06242=1240.660,-56.226,-37.373,-179.908,5.196,148.869
C06243=1240.665,-56.475,-37.360,-179.910,5.196,148.869
C06244=1240.670,-56.726,-37.348,-179.913,5.195,148.870
C06245=1240.675,-56.975,-37.336,-179.915,5.196,148.871
C06246=1240.680,-57.224,-37.323,-179.918,5.196,148.872
C06247=1240.685,-57.473,-37.310,-179.920,5.196,148.873
C06248=1240.691,-57.723,-37.298,-179.923,5.195,148.873
C06249=1240.696,-57.973,-37.286,-179.925,5.196,148.874
C06250=1240.700,-58.223,-37.273,-179.927,5.195,148.875
C06251=1240.706,-58.473,-37.261,-179.930,5.196,148.875
C06252=1240.711,-58.722,-37.248,-179.932,5.195,148.876
C06253=1240.716,-58.972,-37.236,-179.935,5.195,148.877
C06254=1240.721,-59.221,-37.224,-179.937,5.195,148.877
C06255=1240.727,-59.471,-37.211,-179.940,5.194,148.878
C06256=1240.732,-59.721,-37.199,-179.942,5.195,148.879
C06257=1240.737,-59.971,-37.186,-179.945,5.195,148.880
C06258=1240.742,-60.220,-37.174,-179.947,5.195,148.880
C06259=1240.747,-60.470,-37.162,-179.950,5.194,148.881
C06260=1240.752,-60.719,-37.149,-179.952,5.195,148.882
C06261=1240.758,-60.969,-37.137,-179.954,5.194,148.883
C06262=1240.763,-61.218,-37.125,-179.956,5.195,148.883
C06263=1240.768,-61.468,-37.113,-179.959,5.194,148.884
C06264=1240.772,-61.718,-37.101,-179.961,5.194,148.885
C06265=1240.777,-61.967,-37.088,-179.964,5.194,148.885
C06266=1240.783,-62.217,-37.076,-179.966,5.194,148.886
C06267=1240.788,-62.467,-37.064,-179.969,5.194,148.887
C06268=1240.793,-62.717,-37.052,-179.971,5.194,148.888
C06269=1240.798,-62.966,-37.039,-179.974,5.194,148.888
C06270=1240.804,-63.216,-37.027,-179.976,5.194,148.889
C06271=1240.809,-63.465,-37.015,-179.979,5.194,148.890
C06272=1240.814,-63.715,-37.003,-179.981,5.194,148.891
C06273=1240.819,-63.964,-36.991,-179.983,5.194,148.891
C06274=1240.824,-64.214,-36.979,-179.986,5.194,148.892
C06275=1240.829,-64.464,-36.966,-179.988,5.194,148.893
C06276=1240.834,-64.714,-36.954,-179.990,5.194,148.893
C06277=1240.839,-64.963,-36.941,-179.993,5.193,148.894
C06278=1240.844,-65.213,-36.929,-179.995,5.194,148.895
C06279=1240.850,-65.463,-36.918,-179.998,5.193,148.896
C06280=1240.854,-65.712,-36.906,180.000,5.194,148.896
C06281=1240.860,-65.962,-36.894,179.997,5.193,148.897
C06282=1240.865,-66.211,-36.881,179.995,5.194,148.898
C06283=1240.870,-66.461,-36.869,179.992,5.193,148.899
C06284=1240.875,-66.711,-36.857,179.990,5.194,148.899
C06285=1240.880,-66.960,-36.845,179.988,5.193,148.900
C06286=1240.886,-67.210,-36.833,179.985,5.193,148.901
C06287=1240.891,-67.460,-36.821,179.983,5.193,148.901
C06288=1240.896,-67.709,-36.809,179.981,5.193,148.902
C06289=1240.901,-67.959,-36.796,179.978,5.193,148.903
C06290=1240.906,-68.208,-36.785,179.976,5.193,148.904
C06291=1240.911,-68.458,-36.773,179.973,5.193,148.904
C06292=1240.916,-68.708,-36.761,179.971,5.193,148.905
C06293=1240.922,-68.958,-36.749,179.968,5.193,148.906
C06294=1240.927,-69.208,-36.737,179.966,5.193,148.907
C06295=1240.932,-69.457,-36.725,179.963,5.193,148.907
C06296=1240.937,-69.706,-36.713,179.961,5.193,148.908
C06297=1240.943,-69.956,-36.701,179.958,5.193,148.909
C06298=1240.948,-70.206,-36.688,179.956,5.193,148.909
C06299=1240.952,-70.455,-36.677,179.954,5.192,148.910
C06300=1240.958,-70.705,-36.665,179.952,5.193,148.911
C06301=1240.963,-70.955,-36.653,179.949,5.192,148.912
C06302=1240.968,-71.204,-36.641,179.947,5.193,148.912
C06303=1240.973,-71.454,-36.629,179.944,5.192,148.913
C06304=1240.978,-71.704,-36.618,179.942,5.192,148.914
C06305=1240.984,-71.953,-36.605,179.939,5.192,148.914
C06306=1240.988,-72.203,-36.594,179.937,5.193,148.915
C06307=1240.994,-72.453,-36.582,179.934,5.192,148.916
C06308=1240.999,-72.703,-36.570,179.932,5.193,148.917
C06309=1241.004,-72.952,-36.558,179.929,5.192,148.917
C06310=1241.009,-73.202,-36.546,179.927,5.192,148.918
C06311=1241.014,-73.452,-36.534,179.925,5.192,148.919
C06312=1241.019,-73.701,-36.523,179.923,5.192,148.920
C06313=1241.024,-73.972,-36.510,179.920,5.192,148.920
C06314=1241.031,-74.242,-36.497,179.917,5.192,148.921
C06315=1241.036,-74.512,-36.484,179.915,5.192,148.922
C06316=1241.042,-74.782,-36.471,179.912,5.192,148.923
C06317=1241.046,-75.032,-36.459,179.910,5.192,148.923
C06318=1241.052,-75.281,-36.448,179.907,5.191,148.924
C06319=1241.058,-75.531,-36.436,179.905,5.192,148.925
C06320=1241.062,-75.780,-36.424,179.902,5.192,148.926
C06321=1241.068,-76.030,-36.412,179.900,5.192,148.926
C06322=1241.072,-76.280,-36.401,179.897,5.192,148.927
C06323=1241.078,-76.530,-36.389,179.895,5.192,148.928
C06324=1241.083,-76.780,-36.377,179.892,5.191,148.929
C06325=1241.088,-77.029,-36.366,179.890,5.192,148.929
C06326=1241.093,-77.279,-36.354,179.888,5.191,148.930
C06327=1241.098,-77.528,-36.342,179.886,5.192,148.931
C06328=1241.103,-77.778,-36.330,179.883,5.191,148.931
C06329=1241.109,-78.027,-36.318,179.881,5.191,148.932
C06330=1241.114,-78.277,-36.307,179.878,5.191,148.933
C06331=1241.119,-78.527,-36.295,179.876,5.191,148.934
C06332=1241.124,-78.777,-36.284,179.873,5.191,148.934
C06333=1241.129,-79.027,-36.272,179.871,5.191,148.935
C06334=1241.134,-79.276,-36.261,179.868,5.191,148.936
C06335=1241.140,-79.526,-36.249,179.866,5.191,148.937
C06336=1241.145,-79.776,-36.237,179.863,5.191,148.937
C06337=1241.150,-80.026,-36.226,179.861,5.191,148.938
C06338=1241.156,-80.275,-36.214,179.859,5.191,148.939
C06339=1241.160,-80.525,-36.203,179.856,5.191,148.939
C06340=1241.166,-80.774,-36.191,179.854,5.191,148.940
C06341=1241.170,-81.024,-36.180,179.852,5.191,148.941
C06342=1241.176,-81.274,-36.168,179.850,5.191,148.942
C06343=1241.181,-81.524,-36.157,179.847,5.191,148.942
C06344=1241.186,-81.774,-36.145,179.845,5.191,148.943
C06345=1241.191,-82.023,-36.134,179.842,5.191,148.944
C06346=1241.197,-82.272,-36.122,179.840,5.191,148.944
C06347=1241.201,-82.522,-36.111,179.837,5.191,148.945
C06348=1241.207,-82.772,-36.099,179.835,5.191,148.946
C06349=1241.212,-83.022,-36.087,179.833,5.191,148.947
C06350=1241.217,-83.272,-36.076,179.830,5.191,148.947
C06351=1241.222,-83.521,-36.065,179.827,5.191,148.948
C06352=1241.228,-83.770,-36.053,179.825,5.191,148.949
C06353=1241.232,-84.020,-36.041,179.823,5.191,148.950
C06354=1241.237,-84.270,-36.030,179.821,5.191,148.950
C06355=1241.243,-84.520,-36.018,179.818,5.190,148.951
C06356=1241.248,-84.769,-36.007,179.816,5.191,148.952
C06357=1241.253,-85.018,-35.995,179.813,5.190,148.952
C06358=1241.258,-85.268,-35.984,179.811,5.191,148.953
C06359=1241.263,-85.518,-35.972,179.808,5.190,148.954
C06360=1241.268,-85.768,-35.962,179.806,5.191,148.955
C06361=1241.274,-86.018,-35.950,179.804,5.190,148.955
C06362=1241.279,-86.267,-35.939,179.801,5.190,148.956
C06363=1241.284,-86.517,-35.928,179.799,5.190,148.957
C06364=1241.289,-86.767,-35.916,179.797,5.190,148.957
C06365=1241.294,-87.016,-35.904,179.795,5.191,148.958
C06366=1241.300,-87.266,-35.893,179.792,5.190,148.959
C06367=1241.305,-87.516,-35.882,179.790,5.191,148.960
C06368=1241.310,-87.765,-35.871,179.787,5.190,148.960
C06369=1241.315,-88.015,-35.859,179.785,5.191,148.961
C06370=1241.320,-88.264,-35.848,179.782,5.190,148.962
C06371=1241.325,-88.514,-35.837,179.780,5.191,148.963
C06372=1241.331,-88.765,-35.826,179.777,5.190,148.963
C06373=1241.335,-89.014,-35.815,179.775,5.191,148.964
C06374=1241.342,-89.263,-35.803,179.772,5.190,148.965
C06375=1241.346,-89.513,-35.792,179.770,5.190,148.965
C06376=1241.351,-89.763,-35.780,179.768,5.190,148.966
C06377=1241.357,-90.013,-35.769,179.765,5.190,148.967
C06378=1241.362,-90.262,-35.758,179.763,5.190,148.968
C06379=1241.367,-90.512,-35.747,179.761,5.190,148.968
C06380=1241.372,-90.762,-35.735,179.758,5.190,148.969
C06381=1241.377,-91.012,-35.725,179.756,5.190,148.970
C06382=1241.382,-91.261,-35.714,179.754,5.190,148.970
C06383=1241.388,-91.511,-35.702,179.751,5.190,148.971
C06384=1241.392,-91.760,-35.690,179.749,5.190,148.972
C06385=1241.398,-92.010,-35.680,179.746,5.190,148.973
C06386=1241.403,-92.260,-35.669,179.744,5.190,148.973
C06387=1241.408,-92.509,-35.657,179.742,5.190,148.974
C06388=1241.413,-92.760,-35.647,179.740,5.190,148.975
C06389=1241.418,-93.009,-35.636,179.737,5.190,148.975
C06390=1241.424,-93.259,-35.624,179.735,5.190,148.976
C06391=1241.429,-93.509,-35.613,179.732,5.190,148.977
C06392=1241.434,-93.758,-35.602,179.730,5.190,148.978
C06393=1241.439,-94.007,-35.591,179.727,5.190,148.979
C06394=1241.445,-94.258,-35.580,179.725,5.190,148.979
C06395=1241.450,-94.507,-35.569,179.722,5.190,148.980
C06396=1241.455,-94.756,-35.558,179.720,5.190,148.981
C06397=1241.460,-95.007,-35.547,179.718,5.190,148.981
C06398=1241.466,-95.256,-35.535,179.715,5.190,148.982
C06399=1241.471,-95.506,-35.525,179.713,5.190,148.983
C06400=1241.475,-95.756,-35.514,179.710,5.190,148.984
C06401=1241.481,-96.005,-35.503,179.708,5.190,148.984
C06402=1241.486,-96.255,-35.491,179.706,5.190,148.985
C06403=1241.491,-96.505,-35.480,179.704,5.190,148.986
C06404=1241.497,-96.755,-35.470,179.701,5.190,148.986
C06405=1241.501,-97.004,-35.459,179.699,5.190,148.987
C06406=1241.507,-97.254,-35.447,179.696,5.189,148.988
C06407=1241.512,-97.504,-35.437,179.694,5.190,148.988
C06408=1241.517,-97.753,-35.425,179.691,5.189,148.989
C06409=1241.522,-98.003,-35.415,179.689,5.190,148.990
C06410=1241.527,-98.252,-35.404,179.687,5.190,148.991
C06411=1241.532,-98.503,-35.393,179.685,5.190,148.991
C06412=1241.538,-98.752,-35.382,179.682,5.190,148.992
C06413=1241.543,-99.002,-35.371,179.680,5.190,148.993
C06414=1241.548,-99.252,-35.360,179.678,5.190,148.993
C06415=1241.554,-99.501,-35.350,179.675,5.189,148.994
C06416=1241.558,-99.751,-35.338,179.673,5.190,148.995
C06417=1241.564,-100.022,-35.326,179.670,5.189,148.996
C06418=1241.570,-100.293,-35.315,179.668,5.190,148.997
C06419=1241.575,-100.563,-35.303,179.665,5.190,148.997
C06420=1241.581,-100.834,-35.291,179.663,5.190,148.998
C06421=1241.587,-101.084,-35.281,179.660,5.189,148.999
C06422=1241.591,-101.334,-35.270,179.658,5.190,148.999
C06423=1241.597,-101.583,-35.259,179.655,5.189,149.000
C06424=1241.602,-101.833,-35.248,179.653,5.190,149.001
C06425=1241.607,-102.083,-35.237,179.651,5.189,149.002
C06426=1241.612,-102.332,-35.227,179.649,5.190,149.002
C06427=1241.618,-102.583,-35.215,179.646,5.189,149.003
C06428=1241.623,-102.831,-35.204,179.644,5.190,149.004
C06429=1241.628,-103.082,-35.194,179.641,5.189,149.004
C06430=1241.633,-103.331,-35.184,179.639,5.189,149.005
C06431=1241.638,-103.581,-35.172,179.637,5.190,149.006
C06432=1241.643,-103.831,-35.162,179.634,5.189,149.007
C06433=1241.648,-104.080,-35.151,179.632,5.190,149.007
C06434=1241.653,-104.330,-35.140,179.629,5.189,149.008
C06435=1241.659,-104.580,-35.130,179.627,5.190,149.009
C06436=1241.664,-104.829,-35.119,179.625,5.189,149.009
C06437=1241.669,-105.079,-35.109,179.623,5.190,149.010
C06438=1241.674,-105.329,-35.098,179.620,5.189,149.011
C06439=1241.680,-105.578,-35.087,179.618,5.189,149.012
C06440=1241.685,-105.828,-35.077,179.615,5.189,149.012
C06441=1241.690,-106.078,-35.066,179.613,5.189,149.013
C06442=1241.695,-106.328,-35.055,179.610,5.190,149.014
C06443=1241.701,-106.577,-35.045,179.608,5.190,149.015
C06444=1241.706,-106.827,-35.034,179.606,5.190,149.015
C06445=1241.711,-107.076,-35.023,179.603,5.190,149.016
C06446=1241.716,-107.327,-35.013,179.601,5.190,149.017
C06447=1241.721,-107.576,-35.003,179.598,5.189,149.018
C06448=1241.726,-107.826,-34.992,179.596,5.190,149.018
C06449=1241.732,-108.075,-34.981,179.593,5.189,149.019
C06450=1241.737,-108.325,-34.970,179.591,5.190,149.020
C06451=1241.742,-108.575,-34.960,179.589,5.189,149.020
C06452=1241.747,-108.825,-34.950,179.587,5.190,149.021
C06453=1241.753,-109.074,-34.939,179.585,5.190,149.022
C06454=1241.758,-109.324,-34.928,179.582,5.189,149.022
C06455=1241.763,-109.574,-34.918,179.580,5.189,149.023
C06456=1241.768,-109.824,-34.907,179.578,5.189,149.024
C06457=1241.773,-110.073,-34.896,179.575,5.189,149.024
C06458=1241.778,-110.323,-34.886,179.573,5.189,149.025
C06459=1241.784,-110.573,-34.876,179.571,5.189,149.026
C06460=1241.789,-110.823,-34.865,179.568,5.189,149.027
C06461=1241.795,-111.073,-34.855,179.566,5.189,149.027
C06462=1241.799,-111.322,-34.844,179.564,5.190,149.028
C06463=1241.805,-111.572,-34.833,179.561,5.189,149.029
C06464=1241.810,-111.822,-34.823,179.559,5.190,149.029
C06465=1241.816,-112.072,-34.813,179.556,5.189,149.030
C06466=1241.820,-112.321,-34.803,179.554,5.189,149.031
C06467=1241.825,-112.571,-34.792,179.552,5.189,149.032
C06468=1241.831,-112.820,-34.782,179.549,5.189,149.032
C06469=1241.836,-113.070,-34.771,179.547,5.189,149.033
C06470=1241.841,-113.320,-34.761,179.545,5.189,149.034
C06471=1241.846,-113.570,-34.750,179.543,5.190,149.034
C06472=1241.852,-113.820,-34.740,179.540,5.189,149.035
C06473=1241.857,-114.069,-34.730,179.538,5.190,149.036
C06474=1241.862,-114.319,-34.719,179.535,5.189,149.037
C06475=1241.867,-114.569,-34.710,179.533,5.189,149.037
C06476=1241.872,-114.818,-34.698,179.530,5.189,149.038
C06477=1241.878,-115.068,-34.688,179.528,5.189,149.039
C06478=1241.883,-115.317,-34.678,179.526,5.189,149.039
C06479=1241.888,-115.568,-34.667,179.523,5.189,149.040
C06480=1241.894,-115.817,-34.657,179.521,5.190,149.041
C06481=1241.899,-116.067,-34.646,179.519,5.189,149.042
C06482=1241.904,-116.317,-34.637,179.517,5.190,149.042
C06483=1241.909,-116.566,-34.627,179.514,5.189,149.043
C06484=1241.914,-116.816,-34.616,179.512,5.190,149.044
C06485=1241.920,-117.066,-34.606,179.509,5.189,149.044
C06486=1241.925,-117.316,-34.595,179.507,5.189,149.045
C06487=1241.930,-117.565,-34.586,179.504,5.189,149.046
C06488=1241.935,-117.815,-34.575,179.502,5.189,149.047
C06489=1241.940,-118.065,-34.565,179.500,5.190,149.047
C06490=1241.946,-118.315,-34.555,179.497,5.189,149.048
C06491=1241.952,-118.564,-34.544,179.495,5.190,149.049
C06492=1241.956,-118.814,-34.535,179.493,5.189,149.049
C06493=1241.961,-119.064,-34.524,179.491,5.190,149.050
C06494=1241.966,-119.314,-34.514,179.488,5.189,149.051
C06495=1241.972,-119.564,-34.504,179.486,5.189,149.052
C06496=1241.977,-119.813,-34.494,179.484,5.190,149.052
C06497=1241.982,-120.063,-34.483,179.481,5.189,149.053
C06498=1241.987,-120.313,-34.473,179.479,5.189,149.054
C06499=1241.993,-120.562,-34.463,179.477,5.189,149.054
C06500=1241.997,-120.812,-34.453,179.475,5.189,149.055
C06501=1242.003,-121.062,-34.443,179.472,5.189,149.056
C06502=1242.008,-121.311,-34.433,179.470,5.189,149.056
C06503=1242.014,-121.562,-34.423,179.467,5.189,149.057
C06504=1242.019,-121.811,-34.413,179.465,5.189,149.058
C06505=1242.024,-122.061,-34.403,179.463,5.190,149.059
C06506=1242.029,-122.311,-34.392,179.460,5.189,149.059
C06507=1242.034,-122.560,-34.383,179.458,5.189,149.060
C06508=1242.040,-122.810,-34.372,179.456,5.189,149.061
C06509=1242.045,-123.059,-34.362,179.453,5.189,149.061
C06510=1242.050,-123.310,-34.352,179.451,5.189,149.062
C06511=1242.055,-123.559,-34.343,179.449,5.189,149.063
C06512=1242.061,-123.809,-34.333,179.447,5.190,149.064
C06513=1242.066,-124.059,-34.322,179.444,5.189,149.064
C06514=1242.071,-124.309,-34.312,179.442,5.190,149.065
C06515=1242.077,-124.558,-34.302,179.439,5.189,149.066
C06516=1242.082,-124.808,-34.292,179.437,5.190,149.066
C06517=1242.087,-125.058,-34.283,179.434,5.189,149.067
C06518=1242.092,-125.308,-34.272,179.433,5.189,149.068
C06519=1242.098,-125.557,-34.262,179.430,5.189,149.068
C06520=1242.102,-125.807,-34.252,179.428,5.189,149.069
C06521=1241.681,-125.818,-34.287,179.424,5.193,149.071
C06522=1241.676,-125.568,-34.297,179.426,5.192,149.071
C06523=1241.670,-125.318,-34.306,179.428,5.193,149.070
C06524=1241.665,-125.068,-34.317,179.430,5.192,149.069
C06525=1241.660,-124.819,-34.327,179.433,5.193,149.068
C06526=1241.655,-124.569,-34.337,179.435,5.192,149.068
C06527=1241.649,-124.320,-34.347,179.437,5.193,149.067
C06528=1241.644,-124.069,-34.356,179.439,5.193,149.066
C06529=1241.639,-123.820,-34.367,179.442,5.192,149.066
C06530=1241.633,-123.570,-34.377,179.444,5.193,149.065
C06531=1241.629,-123.320,-34.387,179.446,5.192,149.064
C06532=1241.623,-123.071,-34.397,179.449,5.193,149.064
C06533=1241.618,-122.821,-34.407,179.451,5.193,149.063
C06534=1241.613,-122.571,-34.418,179.454,5.193,149.062
C06535=1241.608,-122.321,-34.427,179.456,5.193,149.061
C06536=1241.602,-122.071,-34.437,179.458,5.192,149.061
C06537=1241.596,-121.822,-34.447,179.461,5.193,149.060
C06538=1241.592,-121.572,-34.457,179.463,5.192,149.059
C06539=1241.587,-121.322,-34.467,179.465,5.193,149.059
C06540=1241.581,-121.073,-34.477,179.468,5.192,149.058
C06541=1241.576,-120.823,-34.488,179.470,5.193,149.057
C06542=1241.571,-120.573,-34.498,179.472,5.192,149.056
C06543=1241.566,-120.324,-34.508,179.475,5.193,149.056
C06544=1241.561,-120.074,-34.518,179.477,5.193,149.055
C06545=1241.555,-119.824,-34.529,179.479,5.192,149.054
C06546=1241.550,-119.575,-34.538,179.482,5.193,149.054
C06547=1241.545,-119.324,-34.549,179.483,5.193,149.053
C06548=1241.539,-119.074,-34.558,179.486,5.193,149.052
C06549=1241.534,-118.824,-34.569,179.488,5.193,149.052
C06550=1241.529,-118.575,-34.578,179.491,5.193,149.051
C06551=1241.524,-118.325,-34.589,179.493,5.193,149.050
C06552=1241.519,-118.075,-34.599,179.496,5.193,149.049
C06553=1241.513,-117.826,-34.609,179.498,5.193,149.049
C06554=1241.508,-117.576,-34.619,179.500,5.192,149.048
C06555=1241.503,-117.326,-34.630,179.503,5.193,149.047
C06556=1241.498,-117.077,-34.640,179.505,5.193,149.047
C06557=1241.492,-116.827,-34.650,179.507,5.193,149.046
C06558=1241.487,-116.577,-34.661,179.509,5.193,149.045
C06559=1241.482,-116.328,-34.671,179.512,5.193,149.044
C06560=1241.477,-116.078,-34.682,179.514,5.193,149.044
C06561=1241.472,-115.828,-34.692,179.516,5.192,149.043
C06562=1241.466,-115.579,-34.702,179.519,5.193,149.042
C06563=1241.461,-115.329,-34.713,179.521,5.192,149.042
C06564=1241.456,-115.079,-34.723,179.524,5.193,149.041
C06565=1241.451,-114.829,-34.733,179.526,5.193,149.040
C06566=1241.446,-114.580,-34.743,179.529,5.193,149.039
C06567=1241.440,-114.330,-34.753,179.531,5.193,149.039
C06568=1241.435,-114.080,-34.764,179.533,5.193,149.038
C06569=1241.430,-113.830,-34.774,179.535,5.193,149.037
C06570=1241.425,-113.580,-34.784,179.537,5.192,149.037
C06571=1241.419,-113.330,-34.795,179.540,5.193,149.036
C06572=1241.414,-113.081,-34.806,179.542,5.192,149.035
C06573=1241.409,-112.832,-34.816,179.545,5.193,149.034
C06574=1241.404,-112.582,-34.826,179.547,5.192,149.034
C06575=1241.399,-112.332,-34.836,179.550,5.193,149.033
C06576=1241.393,-112.082,-34.847,179.552,5.193,149.032
C06577=1241.388,-111.832,-34.857,179.555,5.193,149.032
C06578=1241.383,-111.582,-34.867,179.557,5.193,149.031
C06579=1241.378,-111.333,-34.879,179.559,5.192,149.030
C06580=1241.372,-111.083,-34.889,179.561,5.193,149.029
C06581=1241.367,-110.834,-34.899,179.563,5.192,149.029
C06582=1241.362,-110.583,-34.910,179.566,5.193,149.028
C06583=1241.356,-110.334,-34.920,179.568,5.192,149.027
C06584=1241.352,-110.084,-34.931,179.571,5.193,149.027
C06585=1241.346,-109.835,-34.941,179.573,5.193,149.026
C06586=1241.342,-109.585,-34.951,179.576,5.193,149.025
C06587=1241.336,-109.335,-34.962,179.578,5.193,149.024
C06588=1241.331,-109.085,-34.972,179.580,5.193,149.024
C06589=1241.326,-108.836,-34.983,179.583,5.193,149.023
C06590=1241.321,-108.586,-34.994,179.585,5.192,149.022
C06591=1241.315,-108.336,-35.004,179.587,5.193,149.022
C06592=1241.310,-108.086,-35.014,179.589,5.193,149.021
C06593=1241.305,-107.837,-35.025,179.592,5.193,149.020
C06594=1241.300,-107.587,-35.036,179.594,5.193,149.020
C06595=1241.294,-107.337,-35.046,179.596,5.193,149.019
C06596=1241.290,-107.088,-35.057,179.598,5.193,149.018
C06597=1241.284,-106.838,-35.068,179.601,5.193,149.017
C06598=1241.279,-106.588,-35.078,179.603,5.193,149.017
C06599=1241.273,-106.338,-35.088,179.605,5.193,149.016
C06600=1241.269,-106.089,-35.100,179.608,5.193,149.015
C06601=1241.263,-105.839,-35.110,179.610,5.193,149.015
C06602=1241.258,-105.589,-35.120,179.613,5.193,149.014
C06603=1241.253,-105.340,-35.131,179.615,5.193,149.013
C06604=1241.248,-105.090,-35.142,179.618,5.193,149.012
C06605=1241.242,-104.840,-35.152,179.620,5.193,149.012
C06606=1241.238,-104.591,-35.163,179.622,5.193,149.011
C06607=1241.232,-104.340,-35.175,179.625,5.193,149.010
C06608=1241.227,-104.091,-35.186,179.628,5.193,149.009
C06609=1241.222,-103.841,-35.196,179.630,5.193,149.009
C06610=1241.216,-103.591,-35.206,179.632,5.192,149.008
C06611=1241.211,-103.342,-35.218,179.634,5.193,149.007
C06612=1241.206,-103.092,-35.228,179.637,5.193,149.007
C06613=1241.201,-102.842,-35.238,179.639,5.193,149.006
C06614=1241.195,-102.593,-35.249,179.641,5.193,149.005
C06615=1241.190,-102.343,-35.260,179.644,5.193,149.004
C06616=1241.186,-102.093,-35.271,179.646,5.193,149.004
C06617=1241.180,-101.844,-35.281,179.649,5.193,149.003
C06618=1241.175,-101.594,-35.293,179.651,5.193,149.002
C06619=1241.170,-101.344,-35.303,179.654,5.193,149.002
C06620=1241.164,-101.095,-35.315,179.656,5.193,149.001
C06621=1241.159,-100.844,-35.325,179.658,5.193,149.000
C06622=1241.154,-100.574,-35.337,179.660,5.193,148.999
C06623=1241.148,-100.303,-35.348,179.663,5.194,148.999
C06624=1241.142,-100.032,-35.360,179.665,5.193,148.998
C06625=1241.137,-99.762,-35.372,179.668,5.193,148.997
C06626=1241.132,-99.512,-35.383,179.670,5.193,148.996
C06627=1241.126,-99.262,-35.394,179.673,5.193,148.996
C06628=1241.121,-99.013,-35.405,179.675,5.193,148.995
C06629=1241.116,-98.762,-35.416,179.678,5.193,148.994
C06630=1241.111,-98.513,-35.427,179.680,5.193,148.993
C06631=1241.106,-98.263,-35.437,179.683,5.194,148.993
C06632=1241.101,-98.014,-35.448,179.685,5.193,148.992
C06633=1241.095,-97.764,-35.459,179.687,5.193,148.991
C06634=1241.090,-97.514,-35.471,179.690,5.193,148.991
C06635=1241.085,-97.265,-35.481,179.692,5.193,148.990
C06636=1241.080,-97.015,-35.492,179.694,5.193,148.989
C06637=1241.075,-96.765,-35.503,179.696,5.193,148.988
C06638=1241.069,-96.515,-35.514,179.699,5.194,148.988
C06639=1241.064,-96.266,-35.525,179.701,5.193,148.987
C06640=1241.059,-96.016,-35.536,179.704,5.194,148.986
C06641=1241.054,-95.767,-35.547,179.706,5.193,148.986
C06642=1241.049,-95.516,-35.558,179.709,5.194,148.985
C06643=1241.043,-95.266,-35.569,179.711,5.193,148.984
C06644=1241.038,-95.018,-35.580,179.713,5.194,148.983
C06645=1241.033,-94.767,-35.591,179.715,5.193,148.983
C06646=1241.028,-94.518,-35.602,179.718,5.193,148.982
C06647=1241.022,-94.268,-35.613,179.720,5.194,148.981
C06648=1241.017,-94.018,-35.624,179.722,5.193,148.981
C06649=1241.013,-93.769,-35.636,179.725,5.194,148.980
C06650=1241.007,-93.519,-35.646,179.727,5.193,148.979
C06651=1241.002,-93.269,-35.658,179.730,5.194,148.978
C06652=1240.997,-93.019,-35.669,179.732,5.193,148.978
C06653=1240.991,-92.770,-35.679,179.735,5.194,148.977
C06654=1240.986,-92.520,-35.691,179.737,5.193,148.976
C06655=1240.981,-92.270,-35.702,179.740,5.194,148.975
C06656=1240.976,-92.021,-35.713,179.742,5.193,148.975
C06657=1240.971,-91.771,-35.724,179.745,5.194,148.974
C06658=1240.966,-91.521,-35.736,179.747,5.193,148.973
C06659=1240.961,-91.272,-35.747,179.749,5.194,148.973
C06660=1240.955,-91.022,-35.757,179.751,5.194,148.972
C06661=1240.950,-90.772,-35.769,179.754,5.193,148.971
C06662=1240.945,-90.523,-35.780,179.756,5.194,148.970
C06663=1240.940,-90.273,-35.792,179.758,5.193,148.970
C06664=1240.934,-90.023,-35.803,179.761,5.194,148.969
C06665=1240.929,-89.773,-35.814,179.763,5.193,148.968
C06666=1240.925,-89.524,-35.825,179.766,5.194,148.968
C06667=1240.919,-89.275,-35.837,179.768,5.194,148.967
C06668=1240.914,-89.024,-35.847,179.771,5.194,148.966
C06669=1240.909,-88.775,-35.858,179.773,5.194,148.965
C06670=1240.904,-88.525,-35.870,179.775,5.194,148.965
C06671=1240.898,-88.276,-35.881,179.777,5.194,148.964
C06672=1240.893,-88.026,-35.893,179.780,5.194,148.963
C06673=1240.888,-87.776,-35.904,179.782,5.194,148.963
C06674=1240.883,-87.526,-35.915,179.785,5.194,148.962
C06675=1240.878,-87.276,-35.927,179.787,5.194,148.961
C06676=1240.872,-87.027,-35.938,179.790,5.195,148.960
C06677=1240.868,-86.778,-35.949,179.792,5.194,148.960
C06678=1240.862,-86.528,-35.961,179.794,5.193,148.959
C06679=1240.857,-86.277,-35.972,179.797,5.194,148.958
C06680=1240.851,-86.028,-35.983,179.799,5.194,148.957
C06681=1240.847,-85.779,-35.994,179.802,5.194,148.957
C06682=1240.841,-85.529,-36.006,179.804,5.194,148.956
C06683=1240.836,-85.279,-36.018,179.806,5.194,148.955
C06684=1240.832,-85.029,-36.029,179.809,5.194,148.955
C06685=1240.826,-84.780,-36.040,179.811,5.194,148.954
C06686=1240.821,-84.530,-36.052,179.813,5.194,148.953
C06687=1240.815,-84.280,-36.063,179.816,5.194,148.952
C06688=1240.811,-84.030,-36.074,179.818,5.194,148.952
C06689=1240.805,-83.780,-36.086,179.821,5.195,148.951
C06690=1240.800,-83.531,-36.097,179.823,5.194,148.950
C06691=1240.794,-83.281,-36.109,179.826,5.195,148.950
C06692=1240.790,-83.032,-36.120,179.828,5.194,148.949
C06693=1240.785,-82.782,-36.131,179.830,5.195,148.948
C06694=1240.780,-82.532,-36.143,179.832,5.194,148.947
C06695=1240.775,-82.283,-36.155,179.835,5.195,148.947
C06696=1240.769,-82.033,-36.166,179.837,5.195,148.946
C06697=1240.764,-81.784,-36.177,179.840,5.195,148.945
C06698=1240.759,-81.534,-36.189,179.842,5.194,148.944
C06699=1240.754,-81.284,-36.201,179.845,5.195,148.944
C06700=1240.749,-81.034,-36.212,179.847,5.194,148.943
C06701=1240.744,-80.785,-36.224,179.849,5.194,148.942
C06702=1240.739,-80.535,-36.236,179.852,5.195,148.942
C06703=1240.733,-80.286,-36.247,179.854,5.194,148.941
C06704=1240.728,-80.036,-36.258,179.857,5.195,148.940
C06705=1240.722,-79.786,-36.270,179.859,5.194,148.939
C06706=1240.718,-79.536,-36.282,179.861,5.195,148.939
C06707=1240.712,-79.286,-36.294,179.864,5.195,148.938
C06708=1240.708,-79.037,-36.305,179.866,5.195,148.937
C06709=1240.702,-78.787,-36.317,179.868,5.195,148.937
C06710=1240.697,-78.537,-36.328,179.871,5.195,148.936
C06711=1240.691,-78.288,-36.339,179.873,5.195,148.935
C06712=1240.687,-78.039,-36.351,179.876,5.195,148.934
C06713=1240.682,-77.789,-36.363,179.878,5.195,148.934
C06714=1240.676,-77.539,-36.375,179.881,5.195,148.933
C06715=1240.672,-77.289,-36.387,179.883,5.195,148.932
C06716=1240.666,-77.040,-36.398,179.886,5.195,148.931
C06717=1240.661,-76.790,-36.410,179.888,5.195,148.931
C06718=1240.656,-76.540,-36.422,179.891,5.195,148.930
C06719=1240.651,-76.290,-36.433,179.893,5.195,148.929
C06720=1240.646,-76.040,-36.445,179.895,5.195,148.929
C06721=1240.640,-75.792,-36.457,179.897,5.195,148.928
C06722=1240.635,-75.542,-36.469,179.900,5.196,148.927
C06723=1240.630,-75.292,-36.480,179.902,5.195,148.926
C06724=1240.625,-75.042,-36.492,179.905,5.196,148.926
C06725=1240.620,-74.793,-36.503,179.907,5.195,148.925
C06726=1240.615,-74.522,-36.516,179.910,5.195,148.924
C06727=1240.609,-74.253,-36.529,179.912,5.195,148.923
C06728=1240.603,-73.982,-36.543,179.915,5.196,148.923
C06729=1240.597,-73.712,-36.555,179.918,5.196,148.922
C06730=1240.593,-73.462,-36.567,179.920,5.195,148.921
C06731=1240.587,-73.212,-36.579,179.923,5.196,148.920
C06732=1240.582,-72.962,-36.591,179.925,5.196,148.920
C06733=1240.577,-72.714,-36.602,179.928,5.196,148.919
C06734=1240.571,-72.464,-36.614,179.930,5.196,148.918
C06735=1240.566,-72.214,-36.626,179.932,5.196,148.917
C06736=1240.561,-71.964,-36.637,179.934,5.196,148.917
C06737=1240.556,-71.715,-36.650,179.937,5.196,148.916
C06738=1240.551,-71.465,-36.662,179.939,5.196,148.915
C06739=1240.546,-71.215,-36.673,179.942,5.196,148.915
C06740=1240.541,-70.966,-36.685,179.944,5.196,148.914
C06741=1240.535,-70.716,-36.697,179.947,5.197,148.913
C06742=1240.530,-70.466,-36.709,179.949,5.196,148.912
C06743=1240.525,-70.217,-36.721,179.952,5.196,148.912
C06744=1240.520,-69.967,-36.733,179.954,5.196,148.911
C06745=1240.515,-69.717,-36.745,179.957,5.196,148.910
C06746=1240.509,-69.467,-36.757,179.959,5.196,148.909
C06747=1240.505,-69.218,-36.769,179.961,5.197,148.909
C06748=1240.499,-68.969,-36.781,179.963,5.196,148.908
C06749=1240.494,-68.719,-36.793,179.966,5.197,148.907
C06750=1240.489,-68.469,-36.805,179.968,5.196,148.907
C06751=1240.484,-68.220,-36.817,179.971,5.197,148.906
C06752=1240.479,-67.970,-36.829,179.973,5.197,148.905
C06753=1240.474,-67.720,-36.841,179.976,5.197,148.904
C06754=1240.468,-67.470,-36.853,179.978,5.197,148.904
C06755=1240.463,-67.221,-36.866,179.981,5.197,148.903
C06756=1240.458,-66.972,-36.877,179.983,5.197,148.902
C06757=1240.453,-66.722,-36.889,179.986,5.197,148.901
C06758=1240.448,-66.472,-36.902,179.988,5.197,148.901
C06759=1240.443,-66.222,-36.914,179.990,5.197,148.900
C06760=1240.438,-65.972,-36.926,179.993,5.197,148.899
C06761=1240.433,-65.723,-36.938,179.995,5.197,148.899
C06762=1240.428,-65.473,-36.949,179.997,5.197,148.898
C06763=1240.423,-65.223,-36.962,180.000,5.197,148.897
C06764=1240.417,-64.973,-36.974,-179.998,5.197,148.896
C06765=1240.412,-64.724,-36.987,-179.995,5.198,148.896
C06766=1240.407,-64.474,-36.998,-179.993,5.197,148.895
C06767=1240.402,-64.225,-37.010,-179.990,5.197,148.894
C06768=1240.397,-63.975,-37.022,-179.988,5.197,148.893
C06769=1240.392,-63.726,-37.035,-179.985,5.198,148.893
C06770=1240.386,-63.476,-37.047,-179.983,5.197,148.892
C06771=1240.381,-63.227,-37.059,-179.980,5.198,148.891
C06772=1240.376,-62.976,-37.072,-179.978,5.197,148.891
C06773=1240.371,-62.727,-37.084,-179.976,5.198,148.890
C06774=1240.366,-62.477,-37.096,-179.974,5.198,148.889
C06775=1240.361,-62.228,-37.108,-179.971,5.198,148.888
C06776=1240.356,-61.978,-37.120,-179.969,5.198,148.888
C06777=1240.351,-61.729,-37.133,-179.966,5.198,148.887
C06778=1240.345,-61.479,-37.145,-179.964,5.198,148.886
C06779=1240.340,-61.229,-37.157,-179.961,5.198,148.885
C06780=1240.335,-60.980,-37.170,-179.959,5.198,148.885
C06781=1240.330,-60.729,-37.182,-179.956,5.198,148.884
C06782=1240.325,-60.480,-37.195,-179.954,5.198,148.883
C06783=1240.320,-60.230,-37.206,-179.951,5.198,148.883
C06784=1240.315,-59.981,-37.219,-179.949,5.199,148.882
C06785=1240.309,-59.731,-37.231,-179.947,5.199,148.881
C06786=1240.304,-59.482,-37.244,-179.944,5.199,148.880
C06787=1240.299,-59.232,-37.256,-179.942,5.199,148.880
C06788=1240.294,-58.982,-37.268,-179.939,5.199,148.879
C06789=1240.290,-58.733,-37.280,-179.937,5.199,148.878
C06790=1240.285,-58.483,-37.293,-179.935,5.199,148.878
C06791=1240.279,-58.233,-37.305,-179.932,5.199,148.877
C06792=1240.274,-57.984,-37.318,-179.929,5.199,148.876
C06793=1240.269,-57.734,-37.329,-179.927,5.199,148.875
C06794=1240.264,-57.485,-37.342,-179.925,5.199,148.875
C06795=1240.259,-57.235,-37.355,-179.922,5.199,148.874
C06796=1240.254,-56.985,-37.368,-179.920,5.199,148.873
C06797=1240.249,-56.735,-37.379,-179.918,5.199,148.873
C06798=1240.243,-56.486,-37.392,-179.915,5.200,148.872
C06799=1240.238,-56.237,-37.405,-179.913,5.199,148.871
C06800=1240.233,-55.986,-37.417,-179.910,5.200,148.870
C06801=1240.228,-55.737,-37.430,-179.908,5.199,148.870
C06802=1240.223,-55.488,-37.442,-179.905,5.200,148.869
C06803=1240.218,-55.238,-37.454,-179.903,5.199,148.868
C06804=1240.213,-54.988,-37.467,-179.900,5.200,148.867
C06805=1240.207,-54.738,-37.480,-179.898,5.200,148.867
C06806=1240.202,-54.489,-37.493,-179.895,5.200,148.866
C06807=1240.197,-54.239,-37.505,-179.893,5.200,148.865
C06808=1240.192,-53.989,-37.517,-179.891,5.200,148.865
C06809=1240.187,-53.740,-37.530,-179.888,5.201,148.864
C06810=1240.182,-53.490,-37.543,-179.886,5.200,148.863
C06811=1240.177,-53.241,-37.555,-179.883,5.201,148.862
C06812=1240.172,-52.991,-37.567,-179.881,5.200,148.862
C06813=1240.166,-52.741,-37.580,-179.878,5.201,148.861
C06814=1240.162,-52.491,-37.593,-179.876,5.200,148.860
C06815=1240.157,-52.242,-37.605,-179.873,5.201,148.859
C06816=1240.152,-51.993,-37.618,-179.871,5.200,148.859
C06817=1240.146,-51.743,-37.630,-179.869,5.201,148.858
C06818=1240.142,-51.493,-37.643,-179.866,5.201,148.857
C06819=1240.136,-51.243,-37.656,-179.864,5.201,148.857
C06820=1240.131,-50.994,-37.669,-179.861,5.202,148.856
C06821=1240.126,-50.745,-37.681,-179.859,5.201,148.855
C06822=1240.121,-50.495,-37.694,-179.856,5.202,148.854
C06823=1240.116,-50.245,-37.707,-179.854,5.201,148.854
C06824=1240.110,-49.995,-37.719,-179.851,5.202,148.853
C06825=1240.105,-49.746,-37.731,-179.849,5.201,148.852
C06826=1240.100,-49.496,-37.745,-179.846,5.202,148.851
C06827=1240.095,-49.246,-37.758,-179.844,5.201,148.851
C06828=1240.090,-48.997,-37.770,-179.842,5.202,148.850
C06829=1240.085,-48.748,-37.783,-179.840,5.202,148.849
C06830=1240.080,-48.478,-37.796,-179.837,5.202,148.849
C06831=1240.074,-48.208,-37.811,-179.834,5.202,148.848
C06832=1240.069,-47.938,-37.824,-179.832,5.202,148.847
C06833=1240.063,-47.669,-37.838,-179.829,5.202,148.846
C06834=1240.058,-47.419,-37.851,-179.826,5.203,148.846
C06835=1240.053,-47.170,-37.864,-179.824,5.202,148.845
C06836=1240.048,-46.920,-37.876,-179.821,5.203,148.844
C06837=1240.042,-46.671,-37.890,-179.819,5.202,148.843
C06838=1240.037,-46.421,-37.903,-179.816,5.203,148.843
C06839=1240.032,-46.171,-37.915,-179.814,5.203,148.842
C06840=1240.027,-45.922,-37.928,-179.812,5.203,148.841
C06841=1240.023,-45.672,-37.941,-179.809,5.203,148.840
C06842=1240.017,-45.422,-37.954,-179.807,5.203,148.840
C06843=1240.012,-45.173,-37.967,-179.804,5.204,148.839
C06844=1240.007,-44.923,-37.980,-179.802,5.203,148.838
C06845=1240.002,-44.674,-37.992,-179.799,5.204,148.838
C06846=1239.996,-44.424,-38.005,-179.797,5.203,148.837
C06847=1239.992,-44.174,-38.018,-179.794,5.204,148.836
C06848=1239.987,-43.925,-38.031,-179.792,5.203,148.835
C06849=1239.981,-43.675,-38.044,-179.789,5.204,148.835
C06850=1239.976,-43.425,-38.057,-179.787,5.204,148.834
C06851=1239.971,-43.176,-38.070,-179.785,5.204,148.833
C06852=1239.966,-42.926,-38.082,-179.782,5.205,148.832
C06853=1239.961,-42.676,-38.096,-179.780,5.204,148.832
C06854=1239.956,-42.427,-38.108,-179.777,5.205,148.831
C06855=1239.951,-42.177,-38.121,-179.775,5.205,148.830
C06856=1239.945,-41.928,-38.135,-179.772,5.205,148.830
C06857=1239.940,-41.678,-38.148,-179.770,5.204,148.829
C06858=1239.936,-41.428,-38.161,-179.767,5.205,148.828
C06859=1239.931,-41.179,-38.173,-179.765,5.205,148.827
C06860=1239.925,-40.929,-38.187,-179.762,5.205,148.827
C06861=1239.920,-40.679,-38.200,-179.760,5.206,148.826
C06862=1239.915,-40.430,-38.212,-179.758,5.205,148.825
C06863=1239.910,-40.180,-38.227,-179.755,5.206,148.825
C06864=1239.905,-39.931,-38.239,-179.753,5.205,148.824
C06865=1239.900,-39.681,-38.253,-179.750,5.206,148.823
C06866=1239.895,-39.431,-38.265,-179.748,5.206,148.822
C06867=1239.890,-39.182,-38.278,-179.745,5.206,148.821
C06868=1239.884,-38.932,-38.291,-179.743,5.205,148.821
C06869=1239.880,-38.683,-38.305,-179.740,5.206,148.820
C06870=1239.875,-38.433,-38.318,-179.738,5.207,148.819
C06871=1239.869,-38.183,-38.331,-179.736,5.206,148.819
C06872=1239.864,-37.934,-38.344,-179.733,5.207,148.818
C06873=1239.859,-37.684,-38.358,-179.731,5.206,148.817
C06874=1239.854,-37.435,-38.370,-179.728,5.207,148.817
C06875=1239.849,-37.185,-38.383,-179.726,5.207,148.816
C06876=1239.844,-36.935,-38.397,-179.723,5.207,148.815
C06877=1239.839,-36.686,-38.410,-179.721,5.208,148.814
C06878=1239.833,-36.436,-38.423,-179.718,5.207,148.814
C06879=1239.829,-36.186,-38.436,-179.715,5.207,148.813
C06880=1239.823,-35.937,-38.450,-179.713,5.207,148.812
C06881=1239.818,-35.688,-38.463,-179.711,5.208,148.811
C06882=1239.814,-35.438,-38.476,-179.709,5.207,148.811
C06883=1239.808,-35.188,-38.489,-179.706,5.208,148.810
C06884=1239.804,-34.939,-38.503,-179.703,5.208,148.809
C06885=1239.798,-34.689,-38.516,-179.701,5.208,148.809
C06886=1239.793,-34.439,-38.529,-179.699,5.209,148.808
C06887=1239.788,-34.190,-38.543,-179.696,5.208,148.807
C06888=1239.783,-33.940,-38.556,-179.694,5.209,148.807
C06889=1239.777,-33.691,-38.569,-179.691,5.208,148.806
C06890=1239.773,-33.441,-38.583,-179.689,5.209,148.805
C06891=1239.767,-33.192,-38.596,-179.686,5.209,148.804
C06892=1239.763,-32.942,-38.609,-179.684,5.209,148.804
C06893=1239.757,-32.693,-38.623,-179.681,5.209,148.803
C06894=1239.753,-32.443,-38.636,-179.679,5.209,148.802
C06895=1239.747,-32.193,-38.649,-179.676,5.210,148.801
C06896=1239.743,-31.944,-38.663,-179.674,5.210,148.801
C06897=1239.737,-31.694,-38.676,-179.672,5.210,148.800
C06898=1239.733,-31.445,-38.689,-179.669,5.210,148.799
C06899=1239.727,-31.195,-38.703,-179.666,5.210,148.798
C06900=1239.722,-30.946,-38.716,-179.664,5.210,148.798
C06901=1239.717,-30.696,-38.730,-179.662,5.210,148.797
C06902=1239.712,-30.446,-38.743,-179.659,5.210,148.796
C06903=1239.706,-30.197,-38.756,-179.656,5.211,148.796
C06904=1239.701,-29.947,-38.770,-179.654,5.211,148.795
C06905=1239.697,-29.697,-38.784,-179.652,5.211,148.794
C06906=1239.691,-29.448,-38.797,-179.650,5.211,148.794
C06907=1239.687,-29.198,-38.811,-179.647,5.211,148.793
C06908=1239.681,-28.949,-38.824,-179.644,5.212,148.792
C06909=1239.677,-28.699,-38.837,-179.642,5.211,148.791
C06910=1239.671,-28.450,-38.851,-179.639,5.212,148.790
C06911=1239.666,-28.200,-38.865,-179.637,5.211,148.790
C06912=1239.662,-27.950,-38.878,-179.634,5.212,148.789
C06913=1239.656,-27.701,-38.892,-179.632,5.212,148.788
C06914=1239.651,-27.451,-38.905,-179.629,5.212,148.788
C06915=1239.646,-27.202,-38.919,-179.627,5.213,148.787
C06916=1239.641,-26.951,-38.932,-179.625,5.212,148.786
C06917=1239.636,-26.703,-38.946,-179.622,5.213,148.786
C06918=1239.631,-26.453,-38.960,-179.620,5.212,148.785
C06919=1239.626,-26.203,-38.973,-179.617,5.213,148.784
C06920=1239.621,-25.954,-38.987,-179.615,5.213,148.784
C06921=1239.616,-25.704,-39.000,-179.612,5.213,148.783
C06922=1239.611,-25.455,-39.014,-179.609,5.213,148.782
C06923=1239.606,-25.205,-39.028,-179.607,5.213,148.781
C06924=1239.600,-24.955,-39.041,-179.605,5.214,148.780
C06925=1239.596,-24.706,-39.055,-179.602,5.214,148.780
C06926=1239.590,-24.456,-39.068,-179.600,5.214,148.779
C06927=1239.585,-24.207,-39.082,-179.597,5.214,148.778
C06928=1239.581,-23.957,-39.096,-179.595,5.214,148.778
C06929=1239.575,-23.707,-39.109,-179.593,5.215,148.777
C06930=1239.570,-23.458,-39.123,-179.590,5.215,148.776
C06931=1239.565,-23.208,-39.138,-179.588,5.215,148.776
C06932=1239.560,-22.958,-39.151,-179.585,5.215,148.775
C06933=1239.555,-22.709,-39.165,-179.582,5.215,148.774
C06934=1239.549,-22.440,-39.179,-179.580,5.215,148.773
C06935=1239.544,-22.171,-39.194,-179.577,5.216,148.773
C06936=1239.538,-21.901,-39.209,-179.574,5.216,148.772
C06937=1239.533,-21.633,-39.224,-179.572,5.215,148.771
C06938=1239.528,-21.383,-39.238,-179.569,5.216,148.770
C06939=1239.523,-21.133,-39.252,-179.567,5.217,148.770
C06940=1239.517,-20.884,-39.265,-179.565,5.216,148.769
C06941=1239.513,-20.634,-39.279,-179.562,5.217,148.768
C06942=1239.508,-20.385,-39.293,-179.559,5.217,148.767
C06943=1239.502,-20.135,-39.306,-179.557,5.217,148.767
C06944=1239.497,-19.885,-39.321,-179.554,5.217,148.766
C06945=1239.492,-19.636,-39.335,-179.552,5.217,148.765
C06946=1239.488,-19.387,-39.348,-179.549,5.217,148.764
C06947=1239.483,-19.137,-39.363,-179.547,5.218,148.764
C06948=1239.477,-18.887,-39.376,-179.545,5.218,148.763
C06949=1239.472,-18.637,-39.390,-179.542,5.218,148.762
C06950=1239.468,-18.388,-39.404,-179.540,5.218,148.762
C06951=1239.463,-18.139,-39.418,-179.537,5.218,148.761
C06952=1239.458,-17.889,-39.432,-179.535,5.219,148.760
C06953=1239.452,-17.639,-39.445,-179.532,5.219,148.760
C06954=1239.447,-17.390,-39.460,-179.530,5.219,148.759
C06955=1239.442,-17.140,-39.474,-179.527,5.220,148.758
C06956=1239.438,-16.891,-39.488,-179.525,5.219,148.757
C06957=1239.432,-16.642,-39.502,-179.522,5.219,148.757
C06958=1239.427,-16.392,-39.516,-179.520,5.219,148.756
C06959=1239.422,-16.141,-39.529,-179.517,5.220,148.755
C06960=1239.416,-15.892,-39.543,-179.514,5.220,148.755
C06961=1239.411,-15.643,-39.558,-179.512,5.220,148.754
C06962=1239.407,-15.393,-39.572,-179.510,5.220,148.753
C06963=1239.402,-15.144,-39.586,-179.507,5.221,148.752
C06964=1239.397,-14.895,-39.600,-179.505,5.221,148.752
C06965=1239.392,-14.645,-39.614,-179.502,5.221,148.751
C06966=1239.387,-14.395,-39.628,-179.500,5.221,148.750
C06967=1239.382,-14.145,-39.642,-179.498,5.221,148.750
C06968=1239.376,-13.896,-39.656,-179.494,5.222,148.749
C06969=1239.371,-13.647,-39.671,-179.492,5.221,148.748
C06970=1239.366,-13.397,-39.685,-179.490,5.222,148.747
C06971=1239.361,-13.147,-39.699,-179.487,5.222,148.747
C06972=1239.356,-12.897,-39.713,-179.485,5.222,148.746
C06973=1239.351,-12.648,-39.726,-179.482,5.223,148.745
C06974=1239.346,-12.399,-39.740,-179.480,5.222,148.745
C06975=1239.341,-12.149,-39.755,-179.478,5.223,148.744
C06976=1239.337,-11.899,-39.769,-179.475,5.223,148.743
C06977=1239.331,-11.650,-39.783,-179.473,5.223,148.742
C06978=1239.326,-11.400,-39.797,-179.470,5.224,148.742
C06979=1239.321,-11.151,-39.811,-179.468,5.224,148.741
C06980=1239.316,-10.902,-39.826,-179.465,5.224,148.740
C06981=1239.311,-10.652,-39.841,-179.462,5.224,148.739
C06982=1239.306,-10.403,-39.854,-179.460,5.225,148.739
C06983=1239.301,-10.153,-39.869,-179.458,5.224,148.738
C06984=1239.296,-9.904,-39.883,-179.455,5.225,148.737
C06985=1239.291,-9.654,-39.897,-179.452,5.225,148.737
C06986=1239.286,-9.404,-39.912,-179.450,5.225,148.736
C06987=1239.281,-9.154,-39.926,-179.448,5.226,148.735
C06988=1239.276,-8.905,-39.940,-179.445,5.225,148.735
C06989=1239.271,-8.656,-39.954,-179.443,5.226,148.734
C06990=1239.266,-8.406,-39.968,-179.440,5.226,148.733
C06991=1239.261,-8.156,-39.983,-179.438,5.226,148.733
C06992=1239.256,-7.907,-39.997,-179.435,5.227,148.732
C06993=1239.251,-7.657,-40.012,-179.433,5.227,148.731
C06994=1239.246,-7.408,-40.026,-179.431,5.227,148.730
C06995=1239.241,-7.159,-40.040,-179.427,5.227,148.730
C06996=1239.236,-6.909,-40.054,-179.425,5.228,148.729
C06997=1239.231,-6.659,-40.069,-179.423,5.227,148.728
C06998=1239.226,-6.410,-40.083,-179.420,5.228,148.727
C06999=1239.221,-6.160,-40.097,-179.417,5.228,148.727
C07000=1239.216,-5.911,-40.112,-179.415,5.228,148.726
C07001=1239.211,-5.661,-40.126,-179.413,5.229,148.725
C07002=1239.206,-5.411,-40.141,-179.410,5.229,148.725
C07003=1239.200,-5.162,-40.155,-179.408,5.229,148.724
C07004=1239.195,-4.912,-40.169,-179.405,5.229,148.723
C07005=1239.190,-4.663,-40.184,-179.403,5.230,148.723
C07006=1239.185,-4.414,-40.199,-179.401,5.230,148.722
C07007=1239.180,-4.164,-40.213,-179.398,5.230,148.721
C07008=1239.175,-3.914,-40.227,-179.395,5.231,148.721
C07009=1239.171,-3.665,-40.242,-179.393,5.230,148.720
C07010=1239.166,-3.415,-40.257,-179.390,5.231,148.719
C07011=1239.161,-3.166,-40.271,-179.387,5.231,148.718
C07012=1239.155,-2.916,-40.286,-179.385,5.231,148.718
C07013=1239.150,-2.667,-40.300,-179.383,5.231,148.717
C07014=1239.145,-2.417,-40.315,-179.380,5.232,148.716
C07015=1239.140,-2.168,-40.329,-179.378,5.232,148.716
C07016=1239.135,-1.919,-40.344,-179.375,5.232,148.715
C07017=1239.130,-1.669,-40.358,-179.373,5.233,148.714
C07018=1239.125,-1.419,-40.373,-179.371,5.232,148.713
C07019=1239.120,-1.170,-40.388,-179.368,5.233,148.713
C07020=1239.115,-0.920,-40.402,-179.365,5.234,148.712
C07021=1239.110,-0.670,-40.417,-179.363,5.233,148.711
C07022=1239.106,-0.421,-40.432,-179.361,5.234,148.711
C07023=1239.101,-0.172,-40.446,-179.358,5.234,148.710
C07024=1239.095,0.078,-40.461,-179.355,5.234,148.709
C07025=1239.090,0.327,-40.476,-179.353,5.234,148.708
C07026=1239.085,0.577,-40.490,-179.350,5.235,148.708
C07027=1239.080,0.827,-40.504,-179.348,5.234,148.707
C07028=1239.076,1.076,-40.519,-179.345,5.235,148.706
C07029=1239.070,1.326,-40.534,-179.343,5.236,148.706
C07030=1239.065,1.575,-40.549,-179.341,5.235,148.705
C07031=1239.060,1.825,-40.563,-179.338,5.236,148.704
C07032=1239.055,2.075,-40.578,-179.335,5.236,148.704
C07033=1239.050,2.324,-40.593,-179.333,5.236,148.703
C07034=1239.045,2.574,-40.608,-179.330,5.237,148.702
C07035=1239.040,2.823,-40.623,-179.328,5.237,148.702
C07036=1239.035,3.072,-40.637,-179.326,5.237,148.701
C07037=1239.030,3.322,-40.652,-179.323,5.237,148.700
C07038=1239.025,3.591,-40.668,-179.320,5.238,148.699
C07039=1239.020,3.859,-40.684,-179.317,5.238,148.699
C07040=1239.014,4.129,-40.700,-179.315,5.239,148.698
C07041=1239.008,4.397,-40.715,-179.313,5.238,148.697
C07042=1239.004,4.647,-40.730,-179.310,5.239,148.696
C07043=1238.999,4.896,-40.746,-179.307,5.239,148.696
C07044=1238.994,5.146,-40.760,-179.305,5.239,148.695
C07045=1238.989,5.395,-40.775,-179.302,5.239,148.694
C07046=1238.983,5.645,-40.790,-179.299,5.240,148.693
C07047=1238.979,5.894,-40.805,-179.297,5.240,148.693
C07048=1238.974,6.143,-40.820,-179.295,5.240,148.692
C07049=1238.968,6.393,-40.835,-179.292,5.241,148.691
C07050=1238.964,6.643,-40.850,-179.289,5.241,148.691
C07051=1238.959,6.892,-40.864,-179.287,5.241,148.690
C07052=1238.953,7.142,-40.880,-179.285,5.242,148.689
C07053=1238.948,7.391,-40.894,-179.282,5.242,148.689
C07054=1238.944,7.640,-40.909,-179.280,5.242,148.688
C07055=1238.938,7.890,-40.924,-179.277,5.242,148.687
C07056=1238.933,8.140,-40.939,-179.275,5.243,148.687
C07057=1238.928,8.389,-40.954,-179.273,5.243,148.686
C07058=1238.923,8.639,-40.969,-179.270,5.243,148.685
C07059=1238.918,8.888,-40.984,-179.267,5.244,148.685
C07060=1238.914,9.138,-41.000,-179.265,5.244,148.684
C07061=1238.909,9.388,-41.014,-179.262,5.244,148.683
C07062=1238.904,9.637,-41.029,-179.260,5.245,148.682
C07063=1238.899,9.886,-41.044,-179.257,5.245,148.682
C07064=1238.894,10.136,-41.059,-179.255,5.244,148.681
C07065=1238.888,10.385,-41.074,-179.252,5.245,148.680
C07066=1238.884,10.634,-41.089,-179.249,5.246,148.680
C07067=1238.878,10.884,-41.104,-179.247,5.246,148.679
C07068=1238.873,11.133,-41.119,-179.245,5.246,148.678
C07069=1238.869,11.383,-41.134,-179.242,5.246,148.677
C07070=1238.864,11.633,-41.150,-179.239,5.247,148.677
C07071=1238.859,11.882,-41.164,-179.237,5.247,148.676
C07072=1238.853,12.132,-41.180,-179.235,5.247,148.675
C07073=1238.849,12.381,-41.195,-179.232,5.248,148.675
C07074=1238.843,12.631,-41.210,-179.229,5.248,148.674
C07075=1238.838,12.880,-41.225,-179.227,5.248,148.673
C07076=1238.833,13.129,-41.240,-179.225,5.249,148.673
C07077=1238.829,13.379,-41.256,-179.222,5.249,148.672
C07078=1238.824,13.629,-41.271,-179.220,5.249,148.671
C07079=1238.819,13.878,-41.286,-179.217,5.249,148.671
C07080=1238.813,14.128,-41.301,-179.215,5.250,148.670
C07081=1238.809,14.377,-41.316,-179.212,5.251,148.669
C07082=1238.803,14.626,-41.332,-179.210,5.250,148.669
C07083=1238.799,14.876,-41.347,-179.207,5.251,148.668
C07084=1238.793,15.126,-41.362,-179.204,5.251,148.667
C07085=1238.789,15.375,-41.377,-179.202,5.251,148.666
C07086=1238.783,15.624,-41.393,-179.200,5.252,148.666
C07087=1238.779,15.874,-41.408,-179.197,5.252,148.665
C07088=1238.773,16.123,-41.423,-179.194,5.253,148.664
C07089=1238.769,16.373,-41.439,-179.192,5.252,148.664
C07090=1238.764,16.623,-41.453,-179.189,5.253,148.663
C07091=1238.758,16.872,-41.469,-179.187,5.253,148.662
C07092=1238.754,17.121,-41.484,-179.184,5.254,148.661
C07093=1238.748,17.371,-41.500,-179.182,5.254,148.661
C07094=1238.744,17.620,-41.515,-179.179,5.254,148.660
C07095=1238.739,17.870,-41.530,-179.177,5.255,148.659
C07096=1238.733,18.119,-41.546,-179.174,5.255,148.659
C07097=1238.729,18.368,-41.561,-179.172,5.255,148.658
C07098=1238.724,18.618,-41.577,-179.169,5.255,148.657
C07099=1238.719,18.868,-41.592,-179.167,5.256,148.657
C07100=1238.714,19.117,-41.608,-179.164,5.256,148.656
C07101=1238.709,19.366,-41.623,-179.162,5.256,148.655
C07102=1238.704,19.615,-41.638,-179.159,5.257,148.655
C07103=1238.699,19.866,-41.654,-179.157,5.257,148.654
C07104=1238.694,20.115,-41.669,-179.154,5.257,148.653
C07105=1238.689,20.364,-41.685,-179.152,5.258,148.653
C07106=1238.684,20.613,-41.700,-179.149,5.258,148.652
C07107=1238.680,20.863,-41.716,-179.147,5.259,148.651
C07108=1238.674,21.113,-41.731,-179.144,5.259,148.651
C07109=1238.669,21.362,-41.747,-179.142,5.259,148.650
C07110=1238.665,21.612,-41.762,-179.139,5.260,148.649
C07111=1238.659,21.861,-41.778,-179.137,5.260,148.648
C07112=1238.654,22.111,-41.793,-179.134,5.260,148.648
C07113=1238.649,22.360,-41.808,-179.132,5.261,148.647
C07114=1238.645,22.610,-41.824,-179.129,5.261,148.646
C07115=1238.639,22.859,-41.840,-179.126,5.262,148.646
C07116=1238.634,23.109,-41.855,-179.124,5.261,148.645
C07117=1238.629,23.358,-41.870,-179.122,5.262,148.644
C07118=1238.624,23.608,-41.886,-179.119,5.262,148.644
C07119=1238.619,23.857,-41.902,-179.116,5.263,148.643
C07120=1238.614,24.106,-41.917,-179.114,5.263,148.642
C07121=1238.610,24.356,-41.933,-179.112,5.263,148.642
C07122=1238.605,24.605,-41.949,-179.109,5.264,148.641
C07123=1238.599,24.855,-41.965,-179.106,5.264,148.640
C07124=1238.595,25.104,-41.980,-179.104,5.264,148.640
C07125=1238.590,25.354,-41.996,-179.102,5.265,148.639
C07126=1238.584,25.603,-42.011,-179.099,5.265,148.638
C07127=1238.580,25.853,-42.027,-179.096,5.266,148.638
C07128=1238.575,26.102,-42.042,-179.094,5.266,148.637
C07129=1238.570,26.351,-42.059,-179.092,5.266,148.636
C07130=1238.565,26.601,-42.075,-179.089,5.267,148.636
C07131=1238.560,26.851,-42.090,-179.086,5.267,148.635
C07132=1238.554,27.100,-42.106,-179.084,5.268,148.634
C07133=1238.550,27.350,-42.121,-179.082,5.268,148.634
C07134=1238.545,27.599,-42.137,-179.079,5.268,148.633
C07135=1238.540,27.848,-42.153,-179.076,5.269,148.632
C07136=1238.535,28.098,-42.169,-179.074,5.269,148.631
C07137=1238.530,28.348,-42.185,-179.072,5.269,148.631
C07138=1238.525,28.596,-42.200,-179.069,5.270,148.630
C07139=1238.520,28.846,-42.216,-179.066,5.270,148.629
C07140=1238.515,29.096,-42.232,-179.064,5.271,148.629
C07141=1238.510,29.346,-42.248,-179.061,5.271,148.628
C07142=1238.505,29.614,-42.265,-179.059,5.271,148.627
C07143=1238.499,29.883,-42.282,-179.056,5.271,148.626
C07144=1238.494,30.151,-42.299,-179.053,5.272,148.626
C07145=1238.488,30.419,-42.317,-179.051,5.272,148.625
C07146=1238.484,30.669,-42.332,-179.048,5.273,148.624
C07147=1238.479,30.918,-42.347,-179.045,5.273,148.624
C07148=1238.474,31.168,-42.364,-179.043,5.274,148.623
C07149=1238.469,31.417,-42.380,-179.041,5.274,148.622
C07150=1238.464,31.666,-42.395,-179.038,5.274,148.622
C07151=1238.459,31.916,-42.412,-179.035,5.275,148.621
C07152=1238.454,32.165,-42.428,-179.033,5.275,148.620
C07153=1238.449,32.415,-42.444,-179.030,5.276,148.620
C07154=1238.444,32.664,-42.460,-179.028,5.276,148.619
C07155=1238.440,32.914,-42.475,-179.025,5.276,148.618
C07156=1238.434,33.163,-42.491,-179.023,5.277,148.618
C07157=1238.429,33.412,-42.507,-179.020,5.277,148.617
C07158=1238.425,33.662,-42.523,-179.018,5.277,148.616
C07159=1238.420,33.911,-42.539,-179.015,5.278,148.616
C07160=1238.415,34.161,-42.555,-179.013,5.278,148.615
C07161=1238.410,34.410,-42.572,-179.010,5.279,148.614
C07162=1238.405,34.660,-42.588,-179.007,5.280,148.614
C07163=1238.399,34.909,-42.603,-179.005,5.279,148.613
C07164=1238.395,35.159,-42.620,-179.003,5.280,148.612
C07165=1238.390,35.408,-42.635,-179.000,5.280,148.612
C07166=1238.385,35.658,-42.652,-178.997,5.281,148.611
C07167=1238.380,35.907,-42.668,-178.995,5.282,148.610
C07168=1238.375,36.157,-42.684,-178.993,5.281,148.610
C07169=1238.370,36.406,-42.700,-178.990,5.282,148.609
C07170=1238.365,36.656,-42.717,-178.987,5.282,148.608
C07171=1238.360,36.905,-42.732,-178.985,5.283,148.608
C07172=1238.355,37.154,-42.748,-178.982,5.284,148.607
C07173=1238.350,37.404,-42.764,-178.980,5.283,148.606
C07174=1238.345,37.653,-42.781,-178.977,5.284,148.605
C07175=1238.340,37.903,-42.797,-178.975,5.284,148.605
C07176=1238.335,38.152,-42.813,-178.972,5.285,148.604
C07177=1238.331,38.401,-42.830,-178.970,5.286,148.603
C07178=1238.326,38.651,-42.846,-178.967,5.286,148.603
C07179=1238.321,38.900,-42.862,-178.965,5.286,148.602
C07180=1238.316,39.150,-42.878,-178.962,5.286,148.601
C07181=1238.311,39.399,-42.894,-178.960,5.287,148.601
C07182=1238.306,39.649,-42.911,-178.957,5.288,148.600
C07183=1238.300,39.898,-42.927,-178.954,5.288,148.599
C07184=1238.296,40.147,-42.944,-178.952,5.288,148.599
C07185=1238.291,40.397,-42.959,-178.950,5.289,148.598
C07186=1238.286,40.646,-42.976,-178.947,5.289,148.598
C07187=1238.281,40.895,-42.992,-178.945,5.290,148.597
C07188=1238.276,41.145,-43.008,-178.942,5.291,148.596
C07189=1238.271,41.394,-43.025,-178.939,5.291,148.596
C07190=1238.267,41.644,-43.041,-178.937,5.291,148.595
C07191=1238.261,41.893,-43.057,-178.935,5.291,148.594
C07192=1238.256,42.143,-43.074,-178.932,5.292,148.594
C07193=1238.252,42.392,-43.091,-178.929,5.293,148.593
C07194=1238.246,42.642,-43.106,-178.927,5.293,148.592
C07195=1238.242,42.891,-43.123,-178.924,5.294,148.592
C07196=1238.237,43.140,-43.139,-178.922,5.294,148.591
C07197=1238.232,43.389,-43.156,-178.919,5.294,148.590
C07198=1238.227,43.640,-43.172,-178.917,5.295,148.590
C07199=1238.221,43.889,-43.189,-178.914,5.295,148.589
C07200=1238.217,44.138,-43.205,-178.912,5.296,148.588
C07201=1238.212,44.387,-43.221,-178.909,5.296,148.587
C07202=1238.207,44.637,-43.238,-178.907,5.296,148.587
C07203=1238.202,44.886,-43.254,-178.904,5.297,148.586
C07204=1238.197,45.135,-43.271,-178.902,5.297,148.585
C07205=1238.192,45.385,-43.288,-178.899,5.298,148.585
C07206=1238.187,45.634,-43.304,-178.896,5.298,148.584
C07207=1238.183,45.884,-43.320,-178.894,5.299,148.583
C07208=1238.178,46.133,-43.337,-178.892,5.299,148.583
C07209=1238.172,46.382,-43.354,-178.889,5.300,148.582
C07210=1238.168,46.632,-43.370,-178.887,5.300,148.582
C07211=1238.163,46.881,-43.387,-178.884,5.301,148.581
C07212=1238.158,47.131,-43.403,-178.882,5.301,148.580
C07213=1238.153,47.381,-43.420,-178.879,5.302,148.580
C07214=1238.148,47.629,-43.436,-178.876,5.303,148.579
C07215=1238.143,47.879,-43.453,-178.874,5.302,148.578
C07216=1238.139,48.128,-43.470,-178.872,5.303,148.578
C07217=1238.133,48.377,-43.487,-178.869,5.304,148.577
C07218=1238.128,48.627,-43.503,-178.866,5.304,148.576
C07219=1238.124,48.876,-43.520,-178.864,5.305,148.576
C07220=1238.118,49.126,-43.536,-178.861,5.305,148.575
C07221=1238.113,49.376,-43.553,-178.859,5.305,148.574
C07222=1238.109,49.625,-43.569,-178.856,5.306,148.574
C07223=1238.104,49.874,-43.586,-178.854,5.306,148.573
C07224=1238.098,50.124,-43.603,-178.851,5.307,148.572
C07225=1238.094,50.373,-43.620,-178.848,5.307,148.572
C07226=1238.089,50.622,-43.636,-178.846,5.308,148.571
C07227=1238.084,50.872,-43.653,-178.844,5.309,148.570
C07228=1238.079,51.121,-43.670,-178.841,5.309,148.570
C07229=1238.075,51.371,-43.687,-178.839,5.309,148.569
C07230=1238.069,51.620,-43.703,-178.836,5.310,148.568
C07231=1238.064,51.869,-43.720,-178.834,5.310,148.568
C07232=1238.060,52.119,-43.737,-178.831,5.311,148.567
C07233=1238.054,52.368,-43.754,-178.828,5.312,148.566
C07234=1238.050,52.617,-43.770,-178.826,5.312,148.566
C07235=1238.044,52.867,-43.788,-178.823,5.313,148.565
C07236=1238.040,53.117,-43.804,-178.821,5.312,148.564
C07237=1238.035,53.365,-43.821,-178.818,5.313,148.564
C07238=1238.030,53.615,-43.838,-178.816,5.314,148.563
C07239=1238.025,53.865,-43.854,-178.813,5.314,148.562
C07240=1238.021,54.114,-43.871,-178.811,5.315,148.562
C07241=1238.015,54.363,-43.888,-178.808,5.316,148.561
C07242=1238.011,54.612,-43.905,-178.806,5.316,148.561
C07243=1238.005,54.862,-43.923,-178.803,5.317,148.560
C07244=1238.001,55.111,-43.939,-178.801,5.317,148.559
C07245=1237.995,55.361,-43.956,-178.798,5.317,148.559
C07246=1237.990,55.629,-43.974,-178.796,5.318,148.558
C07247=1237.985,55.897,-43.993,-178.793,5.318,148.557
C07248=1237.980,56.166,-44.011,-178.790,5.319,148.556
C07249=1237.974,56.435,-44.029,-178.787,5.319,148.556
C07250=1237.969,56.683,-44.046,-178.785,5.320,148.555
C07251=1237.964,56.933,-44.063,-178.783,5.321,148.555
C07252=1237.960,57.183,-44.080,-178.780,5.321,148.554
C07253=1237.956,57.432,-44.097,-178.777,5.322,148.553
C07254=1237.950,57.681,-44.114,-178.775,5.323,148.553
C07255=1237.945,57.930,-44.131,-178.772,5.323,148.552
C07256=1237.940,58.180,-44.148,-178.769,5.324,148.551
C07257=1237.936,58.429,-44.165,-178.767,5.324,148.551
C07258=1237.931,58.679,-44.183,-178.764,5.325,148.550
C07259=1237.925,58.928,-44.200,-178.762,5.325,148.549
C07260=1237.920,59.177,-44.216,-178.759,5.325,148.549
C07261=1237.915,59.427,-44.233,-178.757,5.326,148.548
C07262=1237.911,59.676,-44.251,-178.755,5.327,148.548
C07263=1237.906,59.926,-44.268,-178.752,5.327,148.547
C07264=1237.901,60.175,-44.285,-178.749,5.328,148.546
C07265=1237.895,60.424,-44.302,-178.747,5.329,148.546
C07266=1237.891,60.673,-44.319,-178.744,5.329,148.545
C07267=1237.886,60.923,-44.336,-178.742,5.330,148.544
C07268=1237.882,61.172,-44.353,-178.739,5.330,148.544
C07269=1237.877,61.422,-44.371,-178.737,5.330,148.543
C07270=1237.871,61.671,-44.388,-178.734,5.331,148.542
C07271=1237.867,61.921,-44.405,-178.732,5.331,148.542
C07272=1237.861,62.169,-44.422,-178.729,5.332,148.541
C07273=1237.857,62.419,-44.439,-178.727,5.333,148.540
C07274=1237.852,62.669,-44.456,-178.724,5.333,148.540
C07275=1237.847,62.918,-44.474,-178.722,5.334,148.539
C07276=1237.842,63.167,-44.491,-178.719,5.335,148.538
C07277=1237.837,63.417,-44.508,-178.716,5.335,148.538
C07278=1237.833,63.666,-44.526,-178.714,5.336,148.537
C07279=1237.828,63.916,-44.543,-178.711,5.336,148.536
C07280=1237.822,64.164,-44.561,-178.708,5.337,148.536
C07281=1237.818,64.414,-44.577,-178.707,5.337,148.535
C07282=1237.812,64.663,-44.595,-178.704,5.338,148.535
C07283=1237.808,64.913,-44.613,-178.702,5.338,148.534
C07284=1237.803,65.162,-44.629,-178.699,5.339,148.533
C07285=1237.798,65.411,-44.647,-178.696,5.339,148.533
C07286=1237.793,65.661,-44.664,-178.694,5.340,148.532
C07287=1237.789,65.910,-44.682,-178.691,5.341,148.531
C07288=1237.784,66.160,-44.699,-178.688,5.341,148.531
C07289=1237.779,66.409,-44.717,-178.686,5.342,148.530
C07290=1237.774,66.658,-44.734,-178.684,5.343,148.530
C07291=1237.769,66.908,-44.752,-178.681,5.343,148.529
C07292=1237.763,67.157,-44.769,-178.678,5.344,148.528
C07293=1237.759,67.406,-44.786,-178.676,5.345,148.528
C07294=1237.754,67.655,-44.803,-178.673,5.345,148.527
C07295=1237.749,67.905,-44.821,-178.670,5.346,148.526
C07296=1237.744,68.154,-44.839,-178.668,5.346,148.526
C07297=1237.740,68.403,-44.856,-178.666,5.346,148.525
C07298=1237.735,68.653,-44.873,-178.664,5.347,148.525
C07299=1237.730,68.902,-44.891,-178.661,5.348,148.524
C07300=1237.725,69.151,-44.909,-178.658,5.348,148.523
C07301=1237.720,69.401,-44.926,-178.656,5.349,148.523
C07302=1237.715,69.650,-44.944,-178.653,5.349,148.522
C07303=1237.710,69.900,-44.961,-178.650,5.350,148.521
C07304=1237.705,70.149,-44.979,-178.648,5.351,148.521
